// TwinCAT 3 PLC project PShEll_UniversalBlocks
// Title: PShEll Universal Blocks
// Company: Precision Systems Engineering
// Author: Control Systems Design Department
// ProjectVersion: 1.0.1.1
// Description: PSE Shell - Automation Software Development Kit
// ProgramVersion: 3.1.4023.0
// libraries:
//   CmpBitmapPool, * (System)
//   JS_MC_REF, * (Jenny Science AG)
//   Recipe Management, * (System)
//   Tc2_EtherCAT, * (Beckhoff Automation GmbH)
//   Tc2_IoFunctions, * (Beckhoff Automation GmbH)
//   Tc2_MC2, * (Beckhoff Automation GmbH)
//   Tc2_Standard, * (Beckhoff Automation GmbH)
//   Tc2_SUPS, * (Beckhoff Automation GmbH)
//   Tc2_System, * (Beckhoff Automation GmbH)
//   Tc2_SystemCX, * (Beckhoff Automation GmbH)
//   Tc2_TcpIp, * (Beckhoff Automation GmbH)
//   Tc2_Utilities, * (Beckhoff Automation GmbH)
//   Tc3_EventLogger, * (Beckhoff Automation GmbH)
//   Tc3_McCollisionAvoidance, * (Beckhoff Automation GmbH)
//   Tc3_McCompensations, * (Beckhoff Automation GmbH)
//   Tc3_McCoordinatedMotion, * (Beckhoff Automation GmbH)
//   Tc3_Module, * (Beckhoff Automation GmbH)
//   Tc3_XTS_Utility, * (Beckhoff Automation GmbH)
//   VisuDialogs, * (System)
//   VisuUserMgmt, * (System)
//   Tc2_Math,3.3.1.0,Beckhoff Automation GmbH
//   VisuSymbols,3.5.10.0,System
// project tree:
//   DUTs/Libs/Alarms/AlarmControler/ E_AlarmControlerState.TcDUT (not stored)
//   DUTs/Libs/Alarms/VisuEvents/ E_EventType.TcDUT (not stored), ST_BaseEvent.TcDUT (not stored), ST_Event.TcDUT (not stored)
//   DUTs/Libs/Axis/Universal Axis/ E_AxisJogDirection.TcDUT (not stored), E_AxisState.TcDUT (not stored), E_AxisStateInit.TcDUT (not stored), E_AxisStatePlcOpen.TcDUT (not stored)
//   DUTs/Libs/BowlFeeder/ E_BowlFeederUnitState.TcDUT, E_BowlFeederUnitStateInit.TcDUT
//   DUTs/Libs/Communication/TcpIp/ E_TcpIpDeviceState.TcDUT (not stored), E_TcpIpDeviceStateRecive.TcDUT (not stored), E_TcpIpDeviceStateSend.TcDUT (not stored), E_TcpIpServerStateRunning.TcDUT (not stored), ST_TcpBufferData.TcDUT (not stored)
//   DUTs/Libs/Cylinder/Universal Cylinder/ E_CylinderError.TcDUT (not stored), E_CylinderState.TcDUT (not stored), E_CylinderStateGo.TcDUT (not stored)
//   DUTs/Libs/Digital Devices/Digital Input/ E_DigitalInputExState.TcDUT (not stored)
//   DUTs/Libs/Digital Devices/Lamp Indicator/ E_LampState.TcDUT (not stored)
//   DUTs/Libs/Fixtures/UniversalFixture/ E_UniversalFixtureConnectionType.TcDUT (not stored), E_UniversalFixtureSampleResult.TcDUT (not stored), E_UniversalFixtureState.TcDUT (not stored), E_UniversalFixtureStateAbort.TcDUT (not stored), E_UniversalFixtureStateInit.TcDUT (not stored), E_UniversalFixtureStateMeasure.TcDUT (not stored), E_UniversalFixtureStateReset.TcDUT (not stored)
//   DUTs/Libs/Platform/Common/ ST_UniversalPlatform.TcDUT (not stored)
//   DUTs/Libs/Platform/Universal Machine/ E_MachineCtrlState.TcDUT (not stored)
//   DUTs/Libs/Platform/Universal Safety/ E_SafetyCtrlState.TcDUT (not stored)
//   DUTs/Libs/Platform/Universal Visu/ E_VisuCtrlAlarmControlState.TcDUT (not stored), E_VisuCtrlAxisImgType.TcDUT (not stored), E_VisuCtrlAxisJogMode.TcDUT (not stored), E_VisuCtrlCylinderImgType.TcDUT (not stored), E_VisuCtrlNavBarState.TcDUT (not stored), E_VisuCtrlPageState.TcDUT, E_VisuCtrlRecipeParameterType.TcDUT (not stored), E_VisuCtrlRecipesManagerState.TcDUT (not stored), E_VisuCtrlRobotImgType.TcDUT (not stored), E_VisuCtrlSingleAxisState.TcDUT (not stored), E_VisuCtrlSingleCylinderState.TcDUT (not stored), E_VisuCtrlSingleRobotState.TcDUT (not stored), E_VisuCtrUniversalMachineState.TcDUT (not stored), ST_VisuCtrlAxisFrame.TcDUT (not stored), ST_VisuCtrlCylinderFrame.TcDUT, ST_VisuCtrlFixtureFrame.TcDUT (not stored), ST_VisuCtrlInputFrame.TcDUT (not stored), ST_VisuCtrlOutputFrame.TcDUT (not stored), ST_VisuCtrlRecipeParameter.TcDUT (not stored), ST_VisuCtrlRecipesManager.TcDUT (not stored), ST_VisuCtrlRobotFrame.TcDUT (not stored), ST_VisuCtrlUnitFrame.TcDUT (not stored)
//   DUTs/Libs/Robots/Mitsubishi/CR800/EtherCAT Registers/ ST_CR800EthercatData.TcDUT (not stored)
//   DUTs/Libs/Robots/Mitsubishi/CR800/ E_CR800Error.TcDUT (not stored), ST_CR800UserDefinedArea.TcDUT (not stored)
//   DUTs/Libs/Robots/Mitsubishi/CR800/StateMachine/ E_CR800State.TcDUT (not stored), E_CR800StateAborting.TcDUT (not stored), E_CR800StateCommandExchange.TcDUT (not stored), E_CR800StateCyclePausing.TcDUT (not stored), E_CR800StateCycleStopping.TcDUT (not stored), E_CR800StateDoingRequest.TcDUT (not stored), E_CR800StateHoming.TcDUT (not stored), E_CR800StateInitializing.TcDUT (not stored), E_CR800StateSendPosition.TcDUT (not stored)
//   DUTs/Libs/Robots/Mitsubishi/ E_RobotActions.TcDUT (not stored), E_RobotSystemActions.TcDUT (not stored)
//   DUTs/Libs/SMC SI Unit/ ST_EX260_SEC1.TcDUT
//   DUTs/Libs/Utilities/CSV Data Exchanger/ E_CSVDataExchangerCountColumnsState.TcDUT (not stored), E_CSVDataExchangerInitState.TcDUT (not stored), E_CSVDataExchangerInsertIntoTableState.TcDUT (not stored), E_CSVDataExchangerSelectAllState.TcDUT (not stored), E_CSVDataExchangerSelectRowState.TcDUT (not stored), E_CSVDataExchangerSetNewPathState.TcDUT (not stored), E_CSVDataExchangerState.TcDUT (not stored), ST_CSV_Record.TcDUT (not stored)
//   DUTs/Libs/Utilities/File Logger/ E_FileLoggerAddLogsState.TcDUT (not stored), E_FileLoggerInitState.TcDUT (not stored), E_FileLoggerSetNewPathState.TcDUT (not stored), E_FileLoggerState.TcDUT (not stored)
//   DUTs/Libs/Utilities/Recipe Manager/ E_RecipesManagerReturns.TcDUT (not stored), E_RecipesManagerState.TcDUT (not stored), E_RecipesManagerStateBackup.TcDUT (not stored), E_RecipesManagerStateCreateRemove.TcDUT (not stored), E_RecipesManagerStateInit.TcDUT (not stored), E_RecipesManagerStateReload.TcDUT (not stored)
//   DUTs/Libs/Utilities/TXT Data Exchanger/ E_TXTDataExchangerAddLogsState.TcDUT (not stored), E_TXTDataExchangerInitState.TcDUT (not stored), E_TXTDataExchangerSearchForFileState.TcDUT (not stored), E_TXTDataExchangerSetNewPathState.TcDUT (not stored), E_TXTDataExchangerState.TcDUT (not stored)
//   DUTs/Libs/Vision/Cognex/ E_CognexCameraGetConnectionStatus.TcDUT (not stored), E_CognexCameraGetExprStatus.TcDUT (not stored), E_CognexCameraGetFileListStatus.TcDUT (not stored), E_CognexCameraGetFileStatus.TcDUT (not stored), E_CognexCameraGetJobStatus.TcDUT (not stored), E_CognexCameraGetOnlineStatus.TcDUT (not stored), E_CognexCameraGetPositionState.TcDUT (not stored), E_CognexCameraGetPositionStatus.TcDUT (not stored), E_CognexCameraGetValueEasyBuilderStatus.TcDUT (not stored), E_CognexCameraGetValueSpreadsheetStatus.TcDUT (not stored), E_CognexCameraGetValuesState.TcDUT (not stored), E_CognexCameraGetValuesStatus.TcDUT (not stored), E_CognexCameraGetValueStatus.TcDUT (not stored), E_CognexCameraImageTriggerStatus.TcDUT (not stored), E_CognexCameraInitState.TcDUT (not stored), E_CognexCameraLoadFileStatus.TcDUT (not stored), E_CognexCameraMethodState.TcDUT (not stored), E_CognexCameraPutLiveStatus.TcDUT (not stored), E_CognexCameraPutPortnumStatus.TcDUT (not stored), E_CognexCameraPutTimeoutStatus.TcDUT (not stored), E_CognexCameraPutUpdateStatus.TcDUT (not stored), E_CognexCameraPutWatchStatus.TcDUT (not stored), E_CognexCameraResetSystemStatus.TcDUT (not stored), E_CognexCameraSetJobStatus.TcDUT (not stored), E_CognexCameraSetOnlineStatus.TcDUT (not stored), E_CognexCameraState.TcDUT (not stored), E_CognexCameraStoreFileStatus.TcDUT (not stored)
//   DUTs/Machine/Machine Control/Batch/ ST_BatchData.TcDUT, ST_BatchPerformacne.TcDUT
//   DUTs/Machine/Machine Control/ E_MachineCtrlStateAbort.TcDUT, E_MachineCtrlStateAuto.TcDUT, E_MachineCtrlStateAutoAOI.TcDUT, E_MachineCtrlStateInit.TcDUT, E_MachineCtrlStateManualToAuto.TcDUT, E_MachineCtrlStateUninitialized.TcDUT
//   DUTs/Machine/Machine Control/Internal/ E_GoldenSampleMeasurementState.TcDUT, E_RotaryTableState.TcDUT
//   DUTs/Machine/Shell API/ ST_Shell.TcDUT (not stored), ST_ShellFlags.TcDUT (not stored), ST_ShellPlatform.TcDUT, ST_ShellRecipeData.TcDUT (not stored)
//   DUTs/Machine/Visu Control/ E_VisuCtrlInitializingPopUpFrameSelector.TcDUT, E_VisuCtrlUninitializedFrameSelector.TcDUT, ST_InitializationFrame.TcDUT, ST_UninitializedSetupFrame.TcDUT, ST_UninitializedStartUpFrame.TcDUT
//   / GlobalTextList.TcGTLO, PlcTask.TcTTO, Visualization Manager.TcVMO (not stored), VISU_TASK.TcTTO
//   GVLs/ GVL.TcGVL
//   POUs/Libs/0_Checks/Checks/ CheckBounds.TcPOU (not stored), CheckDivDInt.TcPOU (not stored), CheckDivLInt.TcPOU (not stored), CheckDivLReal.TcPOU (not stored), CheckDivReal.TcPOU (not stored), CheckPointer.TcPOU (not stored), CheckRangeSigned.TcPOU (not stored), CheckRangeUnsigned.TcPOU (not stored), P_Checks.TcPOU (not stored)
//   POUs/Libs/0_Checks/ GVL_Checks.TcGVL (not stored)
//   POUs/Libs/Alarms/AlarmControler/ FB_AlarmControler.TcPOU (not stored), I_AlarmControler.TcIO (not stored)
//   POUs/Libs/Alarms/VisuEvents/ FB_VisuEventsHandling.TcPOU, LDT_TO_STRING.TcPOU (not stored)
//   POUs/Libs/Analog Devices/Analog Device/ FB_AnalogDevice.TcPOU, I_AnalogDevice.TcIO
//   POUs/Libs/Analog Devices/Analog Output/ FB_AnalogOutput.TcPOU, I_AnalogOutput.TcIO
//   POUs/Libs/Axis/ FB_AxisServo.TcPOU (not stored), FB_UniversalAxis.TcPOU (not stored), I_UniversalAxis.TcIO (not stored)
//   POUs/Libs/Bowl Feeder/ FB_BowlFeeder.TcPOU, I_BowlFeeder.TcIO
//   POUs/Libs/Communication/TcpIp/ FUN_StringToTcpBufferData.TcPOU (not stored), FUN_TcpBufferDataToString.TcPOU (not stored)
//   POUs/Libs/Communication/TcpIp/Tcp Buffer/ FB_TcpBuffer.TcPOU (not stored)
//   POUs/Libs/Communication/TcpIp/Tcp Client/ FB_TcpClient.TcPOU (not stored)
//   POUs/Libs/Communication/TcpIp/Tcp Device/ FB_TcpDevice.TcPOU (not stored), I_TcpDevice.TcIO (not stored)
//   POUs/Libs/Communication/TcpIp/Tcp Server/ FB_TcpServer.TcPOU (not stored)
//   POUs/Libs/Cylinder/Double Coil Cylinder/ FB_DoubleCoilCylinder.TcPOU (not stored), FB_DoubleCoilCylinder2.TcPOU (not stored)
//   POUs/Libs/Cylinder/Single Coil Cylinder/ FB_SingleCoilCylinder.TcPOU (not stored), FB_SingleCoilCylinder2.TcPOU (not stored)
//   POUs/Libs/Cylinder/Universal Cylinder/ FB_UniversalCylinder.TcPOU (not stored), I_UniversalCylinder.TcIO (not stored)
//   POUs/Libs/Digital Devices/Digital Device/ FB_DigitalDevice.TcPOU (not stored), I_DigitalDevice.TcIO (not stored)
//   POUs/Libs/Digital Devices/Digital Input/ FB_DigitalInput.TcPOU (not stored), FB_DigitalInputExt.TcPOU (not stored), I_DigitalInput.TcIO (not stored)
//   POUs/Libs/Digital Devices/Digital Output/ FB_DigitalOutput.TcPOU (not stored), I_DigitalOutput.TcIO (not stored)
//   POUs/Libs/Digital Devices/Lamp Indicator/ FB_Lamp.TcPOU (not stored), I_Lamp.TcIO (not stored)
//   POUs/Libs/Fixtures/ FB_UniversalFixture.TcPOU (not stored), I_UniversalFixture.TcIO (not stored)
//   POUs/Libs/Platform/Universal Machine/ FB_UniversalMachine.TcPOU (not stored), I_UniversalMachine.TcIO (not stored)
//   POUs/Libs/Platform/Universal Safety/ FB_UniversalSafety.TcPOU (not stored), I_UniversalSafety.TcIO (not stored)
//   POUs/Libs/Platform/Universal Visu/ FB_UniversalVisu.TcPOU, F_CloseDialog.TcPOU (not stored), F_OpenDialog.TcPOU (not stored)
//   POUs/Libs/Robots/Mitsubishi/ FB_CR800EtherCAT.TcPOU, I_CR800EtherCAT.TcIO (not stored)
//   POUs/Libs/Utilities/Beckhoff UPS/CX2xxx/ FB_UpsCx2xxx.TcPOU (not stored)
//   POUs/Libs/Utilities/Beckhoff UPS/CX5xxx/ FB_UpsCx50xx.TcPOU (not stored), FB_UpsCx51xx.TcPOU (not stored), FB_UpsCx5xxx.TcPOU (not stored), I_BeckhoffUpsCX5xxx.TcIO (not stored)
//   POUs/Libs/Utilities/Beckhoff UPS/Universal CX/ FB_UniversalCxUps.TcPOU (not stored), I_UniversalCxUps.TcIO (not stored)
//   POUs/Libs/Utilities/CSV Data Exchanger/ FB_CSVDataExchanger.TcPOU (not stored), I_CSVDataExchanger.TcIO (not stored)
//   POUs/Libs/Utilities/ FB_DataSetFifo.TcPOU (excluded from build), FB_DataSetFifo_1.TcPOU
//   POUs/Libs/Utilities/File Logger/ FB_FileLogger.TcPOU (not stored), I_FileLogger.TcIO (not stored)
//   POUs/Libs/Utilities/Math/ FUN_Ceil.TcPOU (not stored)
//   POUs/Libs/Utilities/Recipes Manager/ FB_RecipeParameter.TcPOU (not stored), FB_RecipesControler.TcPOU (not stored), I_RecipeParameter.TcIO (not stored), I_RecipesManager.TcIO (not stored)
//   POUs/Libs/Utilities/StringMerge/ FUN_MergeLongStrings10.TcPOU (not stored), FUN_MergeStrings10.TcPOU (not stored), FUN_MergeStrings3.TcPOU (not stored), FUN_MergeStrings4.TcPOU (not stored), FUN_MergeStrings5.TcPOU (not stored), FUN_MergeStrings6.TcPOU (not stored)
//   POUs/Libs/Utilities/Systemtime to String/ FUN_TimestructToDate.TcPOU (not stored), FUN_TimestructToTime.TcPOU (not stored)
//   POUs/Libs/Utilities/TXT Data Exchanger/ FB_TXTDataExchanger.TcPOU (not stored), I_TXTDataExchanger.TcIO (not stored)
//   POUs/Libs/Vision/Cognex/ FB_CognexCamera.TcPOU (not stored), I_CognexCamera.TcIO (not stored)
//   POUs/Machine/ FB_MachineControl.TcPOU, FB_MachineSafety.TcPOU, FB_VisuControl.TcPOU, I_MachineControl.TcIO, ST_VisuCtrlBowlFeeder.TcDUT
//   POUs/Machine/Module/Robot/ E_AOIRobotActions.TcDUT, E_AOIRobotState.TcDUT, E_AOIRobotStateAbort.TcDUT, E_AOIRobotStateInit.TcDUT, E_EtherCATStatusCheck.TcDUT, FB_Robot.TcPOU, I_AOIRobot.TcIO
//   POUs/Machine/Module/RTCVision/ E_RTCCameraInitState.TcDUT, E_RTCCameraMethodState.TcDUT, E_RTCCameraState.TcDUT, E_VisionJob.TcDUT, E_VisionResult.TcDUT, FB_DoubleTrigger.TcPOU, FB_RTCVision.TcPOU, I_RTCVision.TcIO (excluded from build)
//   POUs/Machine/Visu Control/ F_CloseDialog_1.TcPOU (not stored), F_OpenDialog_1.TcPOU (not stored)
//   POUs/PRG/ PRG_AlarmControl.TcPOU, PRG_FB_BowlFeeder.TcPOU (excluded from build), PRG_MachineControl.TcPOU, PRG_MachineSafety.TcPOU, PRG_RecipesManager.TcPOU (not stored), PRG_VisuControl.TcPOU
//   VISUs/Alarms/ EventTable.TcVIS (not stored), EventTableNew.TcVIS (not stored), SingleEvent.TcVIS (not stored)
//   VISUs/Alarms/Image Pools/ IP_EventSeverity.TcIPO (not stored), IP_EventType.TcIPO (not stored)
//   VISUs/Alarms/Text Lists/ TL_EventServerity.TcTLO (not stored), TL_EventType.TcTLO (not stored)
//   VISUs/Headers/ Header.TcVIS, HeaderWinCE.TcVIS (not stored)
//   VISUs/Headers/Image Pools/ IPHeader.TcIPO (not stored)
//   VISUs/Headers/Text Lists/ TL_HeaderMachineState.TcTLO (not stored)
//   VISUs/ Main.TcVIS
//   VISUs/Manual/Image Pools/ IPAxis.TcIPO (not stored), IPCylinder.TcIPO (not stored), IPRobots.TcIPO (not stored)
//   VISUs/Manual/ SingleAxis.TcVIS, SingleFixture.TcVIS (not stored), SingleAxisJogInching.TcVIS (not stored), SingleAxisJogContinous.TcVIS (not stored), SingleAxisJogInchingModulo.TcVIS (not stored), SingleAxisJogStandardSlow.TcVIS (not stored), SingleAxisJogStandardFlast.TcVIS (not stored), SingleCylinder.TcVIS (not stored), SingleDigitalInput.TcVIS, SingleRobot.TcVIS (not stored), SingleSafeOutput.TcVIS (not stored) (excluded from build), SingleSafeInput.TcVIS (not stored) (excluded from build), SingleDigitalOutput.TcVIS (not stored)
//   VISUs/Manual/Text Lists/ TL_ModeSwitchState.TcTLO (not stored), TL_SingleAxisJogMode.TcTLO (not stored), TL_SingleCylinderState.TcTLO (not stored), TL_SingleAxisState.TcTLO (not stored), TL_SingleRobotState.TcTLO (not stored)
//   VISUs/Navigation/ NavBarAuto.TcVIS, NavBarAuxilary.TcVIS, NavBarEmpty.TcVIS (not stored), NavBarInitializing.TcVIS (not stored), NavBarManual.TcVIS, NavBarUninitialized.TcVIS, NavBarUtilities.TcVIS (not stored)
//   VISUs/Pages/Auto/ AOIBowlFeederFrame.TcVIS, AOIBatchPerformanceFrame.TcVIS, AOIHeaderFrame.TcVIS (excluded from build), AOIHeaderKeySwitchFrame.TcVIS (excluded from build), AOIBatchDataFrame.TcVIS (excluded from build), AOISortStationFrame.TcVIS, PageAuto.TcVIS, ST_SortStationParam.TcDUT
//   VISUs/Pages/Initializing/ InitializingDoorLockOpen.TcVIS, InitializingEStopActive.TcVIS, InitializingFixtureConnectionFailed.TcVIS (excluded from build), InitializingNoFixturesAvailable.TcVIS (excluded from build), InitializingRotaryTablePlaceTrayDialog.TcVIS (excluded from build), InitializingStartSafetySystem.TcVIS, InitializingTrayfeederCourtainBroken.TcVIS (excluded from build), InitializingTrayfeederInterupted.TcVIS (excluded from build), PageInitializing.TcVIS
//   VISUs/Pages/ PageAborting.TcVIS (not stored), PageAlarms.TcVIS, PageManualCylinders.TcVIS (not stored), PageManualRobots.TcVIS (not stored), PageManualInputs.TcVIS (not stored), PageManualAxis.TcVIS (not stored), PageManualOutputs.TcVIS (not stored), PageManualSafety.TcVIS (not stored) (excluded from build), PageReadyInitialized.TcVIS (not stored), PageRecipesManager.TcVIS (not stored), PageReset.TcVIS (not stored), PageSwitchMode.TcVIS (not stored)
//   VISUs/Pages/Uninitialized/ PageUninitialized.TcVIS, UninitializedSetupFrame.TcVIS, UninitializedStartUpFrame.TcVIS
//   VISUs/Recipes/ SingleRecipesParameterTypeBool.TcVIS (not stored), SingleRecipesParameterTypeInteger.TcVIS (not stored), SingleRecipesParameterTypeReal.TcVIS (not stored), SingleRecipesParameterTypeString.TcVIS (not stored)
//   VISUs/Recipes/Text Lists/ TL_RecipesManagerReturns.TcTLO (not stored), TL_RecipesManagerStatus.TcTLO (not stored)
// real-time tasks:
//   TASK PlcTask: cycle T#10ms, priority 20, ADS port 350
//   TASK VISU_TASK: cycle T#100000us, priority 30, ADS port 351
// motion (NC):
//   TASK NC-Task 1 SAF: cycle T#2ms, priority 4, ADS port 501
//   TASK NC-Task 1 SVB: cycle T#10ms, priority 8, ADS port 511
//   AXIS Rotary Table (id 2)
//     General: UnitName=°
//     OtherSettings: AllowMotionCmdToSlave=true
//     encoder EncType=19
//       EncPara: ScaleFactorNumerator=72, ScaleFactorDenominator=10000, MaxCount=#xffffffff
//         Inc: RefSearchInverse=true, RefSyncInverse=false
//     drive DrvType=16
//       DrvPara: MaxCount=#xffffffff, DriveControlDWord=#x00020000
//         Analog: TorqueSetpointScale=10, ScaleFactorActTorque=0.1
//         TimeComp: TaskDelayCycles=1
//     controller CtrType=1
//       CtrPara: PriorControlFactor=1
//         Observer: BandWidth=20
// I/O:
//   DEVICE Device 1 (EtherCAT), AmsNetId 5.127.48.56.2.1
//     Term 1 (EK1200) [EK1200-5000 EtherCAT Power supply (2A E-Bus)]
//       Term 2 (EL6900) [EL6900, TwinSAFE PLC]
//       Term 3 (EL6070-0033) [EL6070-0033 1Ch. Licence key terminal, individual licences]
//       Term 4 (EL1904) [EL1904, 4 Ch. Safety Input 24V, TwinSAFE]
//         modules: Module 1 (FSOES)
//       Term 5 (EL1114) [EL1114 4Ch. Dig. Input 24V, 10µs, Sensor Power]
//       Term 6 (EL1904) [EL1904, 4 Ch. Safety Input 24V, TwinSAFE]
//         modules: Module 1 (FSOES)
//       Term 7 (EL2004) [EL2004 4Ch. Dig. Output 24V, 0.5A]
//       Term 8 (EL2904) [EL2904, 4 Ch. Safety Output 24V, 0.5A, TwinSAFE]
//         modules: Module 1 (FSOES), Module 2 (DO)
//       Term 9 (EL1114) [EL1114 4Ch. Dig. Input 24V, 10µs, Sensor Power]
//       Term 10 (EL4004) [EL4004 4Ch. Ana. Output 0-10V, 12bit]
//       Term 11 (EL1904) [EL1904, 4 Ch. Safety Input 24V, TwinSAFE]
//         modules: Module 1 (FSOES)
//       Term 12 (EL2004) [EL2004 4Ch. Dig. Output 24V, 0.5A]
//       Term 13 (EL2004) [EL2004 4Ch. Dig. Output 24V, 0.5A]
//       Term 14 (EL9410) [EL9410 E-Bus Power Supplier  (Diagnostics)]
//       Term 15 (EL1904) [EL1904, 4 Ch. Safety Input 24V, TwinSAFE]
//         modules: Module 1 (FSOES)
//       Term 16 (EL2004) [EL2004 4Ch. Dig. Output 24V, 0.5A]
//       Term 17 (EL2004) [EL2004 4Ch. Dig. Output 24V, 0.5A]
//       Term 18 (EL2904) [EL2904, 4 Ch. Safety Output 24V, 0.5A, TwinSAFE]
//         modules: Module 1 (FSOES), Module 2 (DO)
//       Term 19 (EL1114) [EL1114 4Ch. Dig. Input 24V, 10µs, Sensor Power]
//       Term 20 (EK1122) [EK1122 2 port EtherCAT junction]
//         Box 21 (CompactCom 40 EtherCAT) [CompactCom 40 EtherCAT]
//           modules: Module 1 (4 Stations:CR800 GPIO_REG_IF)
//         Drive 22 (Ezi-SERVO2 EtherCAT) [Ezi-SERVO2 EtherCAT]
//         Box 23 (EX260-SEC1) [EX260-SEC1 EtherCAT SI Unit (32DO_PNP) Rev1.2]
// variable links:
//   NC-Task 1 SAF/Axes/Rotary Table <-> Device 1 (EtherCAT)/Term 1 (EK1200)/Term 20 (EK1122)/Drive 22 (Ezi-SERVO2 EtherCAT)
//     Drive/Inputs/In/nDcOutputTime <-> InfoData/DcOutputShift
//     Drive/Inputs/In/nState1 <-> CSP Inputs/Status Word
//     Drive/Inputs/In/nState2 <-> CSP Inputs/Status Word @bit 8
//     Drive/Inputs/In/nState4 @bit 1 <-> WcState/InputToggle
//     Drive/Inputs/In/nState4 <-> WcState/WcState
//     Drive/Outputs/Out/nCtrl1 <-> CSP Outputs/Control Word
//     Drive/Outputs/Out/nCtrl2 <-> CSP Outputs/Control Word @bit 8
//     Drive/Outputs/Out/nDataOut1 <-> CSP Outputs/Target Position
//     Enc/Inputs/In/nDataIn1 <-> CSP Inputs/Position Actual Value
//     Enc/Inputs/In/nDataIn3 <-> CSP Inputs/Touch probe 1 positive value
//     Enc/Inputs/In/nDataIn5 <-> CSP Inputs/Touch probe 2 positive value
//     Enc/Inputs/In/nDcInputTime <-> InfoData/DcInputShift
//     Enc/Inputs/In/nState4 @bit 1 <-> WcState/InputToggle
//     Enc/Inputs/In/nState4 <-> WcState/WcState
//     Enc/Inputs/In/nState5 <-> CSP Inputs/Touch probe status
//     Enc/Inputs/In/nState6 <-> CSP Inputs/Touch probe status @bit 8
//     Enc/Outputs/Out/nCtrl5 <-> CSP Outputs/Touch probe function
//     Enc/Outputs/Out/nCtrl6 <-> CSP Outputs/Touch probe function @bit 8
//   PShEll_UniversalBlocks/PShEll_UniversalBlocks Instance <-> Device 1 (EtherCAT)/Term 1 (EK1200)/Term 10 (EL4004)
//     PlcTask Outputs/PRG_MachineControl.fbMachineControler.fbBowlFeeder._aoSetpoint.intAnalogOut <-> AO Outputs Channel 1/Analog output
//   PShEll_UniversalBlocks/PShEll_UniversalBlocks Instance <-> Device 1 (EtherCAT)/Term 1 (EK1200)/Term 13 (EL2004)
//     PlcTask Outputs/PRG_MachineControl.fbMachineControler.fbBowlFeeder.doEnable.bOut <-> Channel 1/Output
//     PlcTask Outputs/PRG_MachineControl.fbMachineControler.fbRobot.doRobotModeSwitch.bOut <-> Channel 3/Output
//   PShEll_UniversalBlocks/PShEll_UniversalBlocks Instance <-> Device 1 (EtherCAT)/Term 1 (EK1200)/Term 16 (EL2004)
//     PlcTask Outputs/PRG_MachineControl.fbMachineControler.doTriggerCam{1..4}.doCam.bOut <-> Channel {1..4}/Output  (4 links)
//   PShEll_UniversalBlocks/PShEll_UniversalBlocks Instance <-> Device 1 (EtherCAT)/Term 1 (EK1200)/Term 17 (EL2004)
//     PlcTask Outputs/PRG_MachineControl.fbMachineControler.doTriggerCam5.doCam.bOut <-> Channel 1/Output
//     PlcTask Outputs/PRG_MachineControl.fbMachineControler.doTriggerCam6.doCam.bOut <-> Channel 2/Output
//     PlcTask Outputs/PRG_MachineControl.fbMachineControler.doTriggerCam7.doCam.bOut <-> Channel 3/Output
//   PShEll_UniversalBlocks/PShEll_UniversalBlocks Instance <-> Device 1 (EtherCAT)/Term 1 (EK1200)/Term 19 (EL1114)
//     PlcTask Inputs/PRG_MachineControl.fbMachineControler.diProductPresenceRobot.bIn <-> Channel 4/Input
//     PlcTask Inputs/PRG_MachineControl.fbMachineControler.fbBowlFeeder.diStatusRelay.bIn <-> Channel 3/Input
//   PShEll_UniversalBlocks/PShEll_UniversalBlocks Instance <-> Device 1 (EtherCAT)/Term 1 (EK1200)/Term 20 (EK1122)/Box 21 (CompactCom 40 EtherCAT)
//     PlcTask Inputs/PRG_MachineControl.fbMachineControler.fbRobot.fbCR800.stCR800EthercatData.arrRegistersInput[6000] <-> Module 1 (4 Stations:CR800 GPIO_REG_IF)/Tx PDO (4 Sta.)/RWr(6000)
//     PlcTask Inputs/PRG_MachineControl.fbMachineControler.fbRobot.fbCR800.stCR800EthercatData.arrRegistersInput[6001] <-> Module 1 (4 Stations:CR800 GPIO_REG_IF)/Tx PDO (4 Sta.)/RWr(6001)
//     PlcTask Inputs/PRG_MachineControl.fbMachineControler.fbRobot.fbCR800.stCR800EthercatData.arrRegistersInput[6002] <-> Module 1 (4 Stations:CR800 GPIO_REG_IF)/Tx PDO (4 Sta.)/RWr(6002)
//     PlcTask Inputs/PRG_MachineControl.fbMachineControler.fbRobot.fbCR800.stCR800EthercatData.arrRegistersInput[6003] <-> Module 1 (4 Stations:CR800 GPIO_REG_IF)/Tx PDO (4 Sta.)/RWr(6003)
//     PlcTask Inputs/PRG_MachineControl.fbMachineControler.fbRobot.fbCR800.stCR800EthercatData.arrRegistersInput[6004] <-> Module 1 (4 Stations:CR800 GPIO_REG_IF)/Tx PDO (4 Sta.)/RWr(6004)
//     PlcTask Inputs/PRG_MachineControl.fbMachineControler.fbRobot.fbCR800.stCR800EthercatData.arrRegistersInput[6005] <-> Module 1 (4 Stations:CR800 GPIO_REG_IF)/Tx PDO (4 Sta.)/RWr(6005)
//     PlcTask Inputs/PRG_MachineControl.fbMachineControler.fbRobot.fbCR800.stCR800EthercatData.arrRegistersInput[6006] <-> Module 1 (4 Stations:CR800 GPIO_REG_IF)/Tx PDO (4 Sta.)/RWr(6006)
//     PlcTask Inputs/PRG_MachineControl.fbMachineControler.fbRobot.fbCR800.stCR800EthercatData.arrRegistersInput[6007] <-> Module 1 (4 Stations:CR800 GPIO_REG_IF)/Tx PDO (4 Sta.)/RWr(6007)
//     PlcTask Inputs/PRG_MachineControl.fbMachineControler.fbRobot.fbCR800.stCR800EthercatData.arrRegistersInput[6008] <-> Module 1 (4 Stations:CR800 GPIO_REG_IF)/Tx PDO (4 Sta.)/RWr(6008)
//     PlcTask Inputs/PRG_MachineControl.fbMachineControler.fbRobot.fbCR800.stCR800EthercatData.arrRegistersInput[6009] <-> Module 1 (4 Stations:CR800 GPIO_REG_IF)/Tx PDO (4 Sta.)/RWr(6009)
//     PlcTask Inputs/PRG_MachineControl.fbMachineControler.fbRobot.fbCR800.stCR800EthercatData.arrRegistersInput[6010] <-> Module 1 (4 Stations:CR800 GPIO_REG_IF)/Tx PDO (4 Sta.)/RWr(6010)
//     PlcTask Inputs/PRG_MachineControl.fbMachineControler.fbRobot.fbCR800.stCR800EthercatData.arrRegistersInput[6011] <-> Module 1 (4 Stations:CR800 GPIO_REG_IF)/Tx PDO (4 Sta.)/RWr(6011)
//     PlcTask Inputs/PRG_MachineControl.fbMachineControler.fbRobot.fbCR800.stCR800EthercatData.arrRegistersInput[6012] <-> Module 1 (4 Stations:CR800 GPIO_REG_IF)/Tx PDO (4 Sta.)/RWr(6012)
//     PlcTask Inputs/PRG_MachineControl.fbMachineControler.fbRobot.fbCR800.stCR800EthercatData.arrRegistersInput[6013] <-> Module 1 (4 Stations:CR800 GPIO_REG_IF)/Tx PDO (4 Sta.)/RWr(6013)
//     PlcTask Inputs/PRG_MachineControl.fbMachineControler.fbRobot.fbCR800.stCR800EthercatData.arrRegistersInput[6014] <-> Module 1 (4 Stations:CR800 GPIO_REG_IF)/Tx PDO (4 Sta.)/RWr(6014)
//     PlcTask Inputs/PRG_MachineControl.fbMachineControler.fbRobot.fbCR800.stCR800EthercatData.arrRegistersInput[6015] <-> Module 1 (4 Stations:CR800 GPIO_REG_IF)/Tx PDO (4 Sta.)/RWr(6015)
//     PlcTask Inputs/PRG_MachineControl.fbMachineControler.fbRobot.fbCR800.stCR800EthercatData.arrRegistersInput[6016] <-> Module 1 (4 Stations:CR800 GPIO_REG_IF)/Tx PDO (4 Sta.)/RWr(6016)
//     PlcTask Inputs/PRG_MachineControl.fbMachineControler.fbRobot.fbCR800.stCR800EthercatData.arrRegistersInput[6017] <-> Module 1 (4 Stations:CR800 GPIO_REG_IF)/Tx PDO (4 Sta.)/RWr(6017)
//     PlcTask Inputs/PRG_MachineControl.fbMachineControler.fbRobot.fbCR800.stCR800EthercatData.arrRegistersInput[6018] <-> Module 1 (4 Stations:CR800 GPIO_REG_IF)/Tx PDO (4 Sta.)/RWr(6018)
//     PlcTask Inputs/PRG_MachineControl.fbMachineControler.fbRobot.fbCR800.stCR800EthercatData.arrRegistersInput[6019] <-> Module 1 (4 Stations:CR800 GPIO_REG_IF)/Tx PDO (4 Sta.)/RWr(6019)
//     PlcTask Inputs/PRG_MachineControl.fbMachineControler.fbRobot.fbCR800.stCR800EthercatData.arrRegistersInput[6020] <-> Module 1 (4 Stations:CR800 GPIO_REG_IF)/Tx PDO (4 Sta.)/RWr(6020)
//     PlcTask Inputs/PRG_MachineControl.fbMachineControler.fbRobot.fbCR800.stCR800EthercatData.arrRegistersInput[6021] <-> Module 1 (4 Stations:CR800 GPIO_REG_IF)/Tx PDO (4 Sta.)/RWr(6021)
//     PlcTask Inputs/PRG_MachineControl.fbMachineControler.fbRobot.fbCR800.stCR800EthercatData.arrRegistersInput[6022] <-> Module 1 (4 Stations:CR800 GPIO_REG_IF)/Tx PDO (4 Sta.)/RWr(6022)
//     PlcTask Inputs/PRG_MachineControl.fbMachineControler.fbRobot.fbCR800.stCR800EthercatData.arrRegistersInput[6023] <-> Module 1 (4 Stations:CR800 GPIO_REG_IF)/Tx PDO (4 Sta.)/RWr(6023)
//     PlcTask Inputs/PRG_MachineControl.fbMachineControler.fbRobot.fbCR800.stCR800EthercatData.arrRegistersInput[6024] <-> Module 1 (4 Stations:CR800 GPIO_REG_IF)/Tx PDO (4 Sta.)/RWr(6024)
//     PlcTask Inputs/PRG_MachineControl.fbMachineControler.fbRobot.fbCR800.stCR800EthercatData.arrRegistersInput[6025] <-> Module 1 (4 Stations:CR800 GPIO_REG_IF)/Tx PDO (4 Sta.)/RWr(6025)
//     PlcTask Inputs/PRG_MachineControl.fbMachineControler.fbRobot.fbCR800.stCR800EthercatData.arrRegistersInput[6026] <-> Module 1 (4 Stations:CR800 GPIO_REG_IF)/Tx PDO (4 Sta.)/RWr(6026)
//     PlcTask Inputs/PRG_MachineControl.fbMachineControler.fbRobot.fbCR800.stCR800EthercatData.arrRegistersInput[6027] <-> Module 1 (4 Stations:CR800 GPIO_REG_IF)/Tx PDO (4 Sta.)/RWr(6027)
//     PlcTask Inputs/PRG_MachineControl.fbMachineControler.fbRobot.fbCR800.stCR800EthercatData.arrRegistersInput[6028] <-> Module 1 (4 Stations:CR800 GPIO_REG_IF)/Tx PDO (4 Sta.)/RWr(6028)
//     PlcTask Inputs/PRG_MachineControl.fbMachineControler.fbRobot.fbCR800.stCR800EthercatData.arrRegistersInput[6029] <-> Module 1 (4 Stations:CR800 GPIO_REG_IF)/Tx PDO (4 Sta.)/RWr(6029)
//     PlcTask Inputs/PRG_MachineControl.fbMachineControler.fbRobot.fbCR800.stCR800EthercatData.arrRegistersInput[6030] <-> Module 1 (4 Stations:CR800 GPIO_REG_IF)/Tx PDO (4 Sta.)/RWr(6030)
//     PlcTask Inputs/PRG_MachineControl.fbMachineControler.fbRobot.fbCR800.stCR800EthercatData.arrRegistersInput[6031] <-> Module 1 (4 Stations:CR800 GPIO_REG_IF)/Tx PDO (4 Sta.)/RWr(6031)
//     PlcTask Inputs/PRG_MachineControl.fbMachineControler.fbRobot.fbCR800.stCR800EthercatData.arrRegistersInput[6032] <-> Module 1 (4 Stations:CR800 GPIO_REG_IF)/Tx PDO (4 Sta.)/RWr(6032)
//     PlcTask Inputs/PRG_MachineControl.fbMachineControler.fbRobot.fbCR800.stCR800EthercatData.arrRegistersInput[6033] <-> Module 1 (4 Stations:CR800 GPIO_REG_IF)/Tx PDO (4 Sta.)/RWr(6033)
//     PlcTask Inputs/PRG_MachineControl.fbMachineControler.fbRobot.fbCR800.stCR800EthercatData.arrRegistersInput[6034] <-> Module 1 (4 Stations:CR800 GPIO_REG_IF)/Tx PDO (4 Sta.)/RWr(6034)
//     PlcTask Inputs/PRG_MachineControl.fbMachineControler.fbRobot.fbCR800.stCR800EthercatData.arrRegistersInput[6035] <-> Module 1 (4 Stations:CR800 GPIO_REG_IF)/Tx PDO (4 Sta.)/RWr(6035)
//     PlcTask Inputs/PRG_MachineControl.fbMachineControler.fbRobot.fbCR800.stCR800EthercatData.arrRegistersInput[6036] <-> Module 1 (4 Stations:CR800 GPIO_REG_IF)/Tx PDO (4 Sta.)/RWr(6036)
//     PlcTask Inputs/PRG_MachineControl.fbMachineControler.fbRobot.fbCR800.stCR800EthercatData.arrRegistersInput[6037] <-> Module 1 (4 Stations:CR800 GPIO_REG_IF)/Tx PDO (4 Sta.)/RWr(6037)
//     PlcTask Inputs/PRG_MachineControl.fbMachineControler.fbRobot.fbCR800.stCR800EthercatData.arrRegistersInput[6038] <-> Module 1 (4 Stations:CR800 GPIO_REG_IF)/Tx PDO (4 Sta.)/RWr(6038)
//     PlcTask Inputs/PRG_MachineControl.fbMachineControler.fbRobot.fbCR800.stCR800EthercatData.arrRegistersInput[6039] <-> Module 1 (4 Stations:CR800 GPIO_REG_IF)/Tx PDO (4 Sta.)/RWr(6039)
//     PlcTask Inputs/PRG_MachineControl.fbMachineControler.fbRobot.fbCR800.stCR800EthercatData.arrRegistersInput[6040] <-> Module 1 (4 Stations:CR800 GPIO_REG_IF)/Tx PDO (4 Sta.)/RWr(6040)
//     PlcTask Inputs/PRG_MachineControl.fbMachineControler.fbRobot.fbCR800.stCR800EthercatData.arrRegistersInput[6041] <-> Module 1 (4 Stations:CR800 GPIO_REG_IF)/Tx PDO (4 Sta.)/RWr(6041)
//     PlcTask Inputs/PRG_MachineControl.fbMachineControler.fbRobot.fbCR800.stCR800EthercatData.arrRegistersInput[6042] <-> Module 1 (4 Stations:CR800 GPIO_REG_IF)/Tx PDO (4 Sta.)/RWr(6042)
//     PlcTask Inputs/PRG_MachineControl.fbMachineControler.fbRobot.fbCR800.stCR800EthercatData.arrRegistersInput[6043] <-> Module 1 (4 Stations:CR800 GPIO_REG_IF)/Tx PDO (4 Sta.)/RWr(6043)
//     PlcTask Inputs/PRG_MachineControl.fbMachineControler.fbRobot.fbCR800.stCR800EthercatData.arrRegistersInput[6044] <-> Module 1 (4 Stations:CR800 GPIO_REG_IF)/Tx PDO (4 Sta.)/RWr(6044)
//     PlcTask Inputs/PRG_MachineControl.fbMachineControler.fbRobot.fbCR800.stCR800EthercatData.arrRegistersInput[6045] <-> Module 1 (4 Stations:CR800 GPIO_REG_IF)/Tx PDO (4 Sta.)/RWr(6045)
//     PlcTask Inputs/PRG_MachineControl.fbMachineControler.fbRobot.fbCR800.stCR800EthercatData.arrRegistersInput[6046] <-> Module 1 (4 Stations:CR800 GPIO_REG_IF)/Tx PDO (4 Sta.)/RWr(6046)
//     PlcTask Inputs/PRG_MachineControl.fbMachineControler.fbRobot.fbCR800.stCR800EthercatData.arrRegistersInput[6047] <-> Module 1 (4 Stations:CR800 GPIO_REG_IF)/Tx PDO (4 Sta.)/RWr(6047)
//     PlcTask Inputs/PRG_MachineControl.fbMachineControler.fbRobot.fbCR800.stCR800EthercatData.arrRegistersInput[6048] <-> Module 1 (4 Stations:CR800 GPIO_REG_IF)/Tx PDO (4 Sta.)/RWr(6048)
//     PlcTask Inputs/PRG_MachineControl.fbMachineControler.fbRobot.fbCR800.stCR800EthercatData.arrRegistersInput[6049] <-> Module 1 (4 Stations:CR800 GPIO_REG_IF)/Tx PDO (4 Sta.)/RWr(6049)
//     PlcTask Inputs/PRG_MachineControl.fbMachineControler.fbRobot.fbCR800.stCR800EthercatData.arrRegistersInput[6050] <-> Module 1 (4 Stations:CR800 GPIO_REG_IF)/Tx PDO (4 Sta.)/RWr(6050)
//     PlcTask Inputs/PRG_MachineControl.fbMachineControler.fbRobot.fbCR800.stCR800EthercatData.arrRegistersInput[6051] <-> Module 1 (4 Stations:CR800 GPIO_REG_IF)/Tx PDO (4 Sta.)/RWr(6051)
//     PlcTask Inputs/PRG_MachineControl.fbMachineControler.fbRobot.fbCR800.stCR800EthercatData.arrRegistersInput[6052] <-> Module 1 (4 Stations:CR800 GPIO_REG_IF)/Tx PDO (4 Sta.)/RWr(6052)
//     PlcTask Inputs/PRG_MachineControl.fbMachineControler.fbRobot.fbCR800.stCR800EthercatData.arrRegistersInput[6053] <-> Module 1 (4 Stations:CR800 GPIO_REG_IF)/Tx PDO (4 Sta.)/RWr(6053)
//     PlcTask Inputs/PRG_MachineControl.fbMachineControler.fbRobot.fbCR800.stCR800EthercatData.arrRegistersInput[6054] <-> Module 1 (4 Stations:CR800 GPIO_REG_IF)/Tx PDO (4 Sta.)/RWr(6054)
//     PlcTask Inputs/PRG_MachineControl.fbMachineControler.fbRobot.fbCR800.stCR800EthercatData.arrRegistersInput[6055] <-> Module 1 (4 Stations:CR800 GPIO_REG_IF)/Tx PDO (4 Sta.)/RWr(6055)
//     PlcTask Inputs/PRG_MachineControl.fbMachineControler.fbRobot.fbCR800.stCR800EthercatData.arrRegistersInput[6056] <-> Module 1 (4 Stations:CR800 GPIO_REG_IF)/Tx PDO (4 Sta.)/RWr(6056)
//     PlcTask Inputs/PRG_MachineControl.fbMachineControler.fbRobot.fbCR800.stCR800EthercatData.arrRegistersInput[6057] <-> Module 1 (4 Stations:CR800 GPIO_REG_IF)/Tx PDO (4 Sta.)/RWr(6057)
//     PlcTask Inputs/PRG_MachineControl.fbMachineControler.fbRobot.fbCR800.stCR800EthercatData.arrRegistersInput[6058] <-> Module 1 (4 Stations:CR800 GPIO_REG_IF)/Tx PDO (4 Sta.)/RWr(6058)
//     PlcTask Inputs/PRG_MachineControl.fbMachineControler.fbRobot.fbCR800.stCR800EthercatData.arrRegistersInput[6059] <-> Module 1 (4 Stations:CR800 GPIO_REG_IF)/Tx PDO (4 Sta.)/RWr(6059)
//     PlcTask Inputs/PRG_MachineControl.fbMachineControler.fbRobot.fbCR800.stCR800EthercatData.arrRegistersInput[6060] <-> Module 1 (4 Stations:CR800 GPIO_REG_IF)/Tx PDO (4 Sta.)/RWr(6060)
//     PlcTask Inputs/PRG_MachineControl.fbMachineControler.fbRobot.fbCR800.stCR800EthercatData.arrRegistersInput[6061] <-> Module 1 (4 Stations:CR800 GPIO_REG_IF)/Tx PDO (4 Sta.)/RWr(6061)
//     PlcTask Inputs/PRG_MachineControl.fbMachineControler.fbRobot.fbCR800.stCR800EthercatData.arrRegistersInput[6062] <-> Module 1 (4 Stations:CR800 GPIO_REG_IF)/Tx PDO (4 Sta.)/RWr(6062)
//     PlcTask Inputs/PRG_MachineControl.fbMachineControler.fbRobot.fbCR800.stCR800EthercatData.arrRegistersInput[6063] <-> Module 1 (4 Stations:CR800 GPIO_REG_IF)/Tx PDO (4 Sta.)/RWr(6063)
//     PlcTask Inputs/PRG_MachineControl.fbMachineControler.fbRobot.fbCR800.stCR800EthercatData.arrRegistersInput[6064] <-> Module 1 (4 Stations:CR800 GPIO_REG_IF)/Tx PDO (4 Sta.)/RWr(6064)
//     PlcTask Inputs/PRG_MachineControl.fbMachineControler.fbRobot.fbCR800.stCR800EthercatData.arrRegistersInput[6065] <-> Module 1 (4 Stations:CR800 GPIO_REG_IF)/Tx PDO (4 Sta.)/RWr(6065)
//     PlcTask Inputs/PRG_MachineControl.fbMachineControler.fbRobot.fbCR800.stCR800EthercatData.arrRegistersInput[6066] <-> Module 1 (4 Stations:CR800 GPIO_REG_IF)/Tx PDO (4 Sta.)/RWr(6066)
//     PlcTask Inputs/PRG_MachineControl.fbMachineControler.fbRobot.fbCR800.stCR800EthercatData.arrRegistersInput[6067] <-> Module 1 (4 Stations:CR800 GPIO_REG_IF)/Tx PDO (4 Sta.)/RWr(6067)
//     PlcTask Inputs/PRG_MachineControl.fbMachineControler.fbRobot.fbCR800.stCR800EthercatData.arrRegistersInput[6068] <-> Module 1 (4 Stations:CR800 GPIO_REG_IF)/Tx PDO (4 Sta.)/RWr(6068)
//     PlcTask Inputs/PRG_MachineControl.fbMachineControler.fbRobot.fbCR800.stCR800EthercatData.arrRegistersInput[6069] <-> Module 1 (4 Stations:CR800 GPIO_REG_IF)/Tx PDO (4 Sta.)/RWr(6069)
//     PlcTask Inputs/PRG_MachineControl.fbMachineControler.fbRobot.fbCR800.stCR800EthercatData.arrRegistersInput[6070] <-> Module 1 (4 Stations:CR800 GPIO_REG_IF)/Tx PDO (4 Sta.)/RWr(6070)
//     PlcTask Inputs/PRG_MachineControl.fbMachineControler.fbRobot.fbCR800.stCR800EthercatData.arrRegistersInput[6071] <-> Module 1 (4 Stations:CR800 GPIO_REG_IF)/Tx PDO (4 Sta.)/RWr(6071)
//     PlcTask Inputs/PRG_MachineControl.fbMachineControler.fbRobot.fbCR800.stCR800EthercatData.arrRegistersInput[6072] <-> Module 1 (4 Stations:CR800 GPIO_REG_IF)/Tx PDO (4 Sta.)/RWr(6072)
//     PlcTask Inputs/PRG_MachineControl.fbMachineControler.fbRobot.fbCR800.stCR800EthercatData.arrRegistersInput[6075] <-> Module 1 (4 Stations:CR800 GPIO_REG_IF)/Tx PDO (4 Sta.)/RWr(6075)
//     PlcTask Inputs/PRG_MachineControl.fbMachineControler.fbRobot.fbCR800.stCR800EthercatData.arrRegistersInput[6076] <-> Module 1 (4 Stations:CR800 GPIO_REG_IF)/Tx PDO (4 Sta.)/RWr(6076)
//     PlcTask Inputs/PRG_MachineControl.fbMachineControler.fbRobot.fbCR800.stCR800EthercatData.arrRegistersInput[6077] <-> Module 1 (4 Stations:CR800 GPIO_REG_IF)/Tx PDO (4 Sta.)/RWr(6077)
//     PlcTask Inputs/PRG_MachineControl.fbMachineControler.fbRobot.fbCR800.stCR800EthercatData.arrRegistersInput[6078] <-> Module 1 (4 Stations:CR800 GPIO_REG_IF)/Tx PDO (4 Sta.)/RWr(6078)
//     PlcTask Inputs/PRG_MachineControl.fbMachineControler.fbRobot.fbCR800.stCR800EthercatData.arrRegistersInput[6079] <-> Module 1 (4 Stations:CR800 GPIO_REG_IF)/Tx PDO (4 Sta.)/RWr(6079)
//     PlcTask Inputs/PRG_MachineControl.fbMachineControler.fbRobot.fbCR800.stCR800EthercatData.arrRegistersInput[6080] <-> Module 1 (4 Stations:CR800 GPIO_REG_IF)/Tx PDO (4 Sta.)/RWr(6080)
//     PlcTask Inputs/PRG_MachineControl.fbMachineControler.fbRobot.fbCR800.stCR800EthercatData.arrRegistersInput[6081] <-> Module 1 (4 Stations:CR800 GPIO_REG_IF)/Tx PDO (4 Sta.)/RWr(6081)
//     PlcTask Inputs/PRG_MachineControl.fbMachineControler.fbRobot.fbCR800.stCR800EthercatData.arrRegistersInput[6082] <-> Module 1 (4 Stations:CR800 GPIO_REG_IF)/Tx PDO (4 Sta.)/RWr(6082)
//     PlcTask Inputs/PRG_MachineControl.fbMachineControler.fbRobot.fbCR800.stCR800EthercatData.arrRegistersInput[6083] <-> Module 1 (4 Stations:CR800 GPIO_REG_IF)/Tx PDO (4 Sta.)/RWr(6083)
//     PlcTask Inputs/PRG_MachineControl.fbMachineControler.fbRobot.fbCR800.stCR800EthercatData.arrRegistersInput[6084] <-> Module 1 (4 Stations:CR800 GPIO_REG_IF)/Tx PDO (4 Sta.)/RWr(6084)
//     PlcTask Inputs/PRG_MachineControl.fbMachineControler.fbRobot.fbCR800.stCR800EthercatData.arrRegistersInput[6085] <-> Module 1 (4 Stations:CR800 GPIO_REG_IF)/Tx PDO (4 Sta.)/RWr(6085)
//     PlcTask Inputs/PRG_MachineControl.fbMachineControler.fbRobot.fbCR800.stCR800EthercatData.arrRegistersInput[6086] <-> Module 1 (4 Stations:CR800 GPIO_REG_IF)/Tx PDO (4 Sta.)/RWr(6086)
//     PlcTask Inputs/PRG_MachineControl.fbMachineControler.fbRobot.fbCR800.stCR800EthercatData.arrRegistersInput[6087] <-> Module 1 (4 Stations:CR800 GPIO_REG_IF)/Tx PDO (4 Sta.)/RWr(6087)
//     PlcTask Inputs/PRG_MachineControl.fbMachineControler.fbRobot.fbCR800.stCR800EthercatData.arrRegistersInput[6088] <-> Module 1 (4 Stations:CR800 GPIO_REG_IF)/Tx PDO (4 Sta.)/RWr(6088)
//     PlcTask Inputs/PRG_MachineControl.fbMachineControler.fbRobot.fbCR800.stCR800EthercatData.arrRegistersInput[6089] <-> Module 1 (4 Stations:CR800 GPIO_REG_IF)/Tx PDO (4 Sta.)/RWr(6089)
//     PlcTask Inputs/PRG_MachineControl.fbMachineControler.fbRobot.fbCR800.stCR800EthercatData.arrRegistersInput[6090] <-> Module 1 (4 Stations:CR800 GPIO_REG_IF)/Tx PDO (4 Sta.)/RWr(6090)
//     PlcTask Inputs/PRG_MachineControl.fbMachineControler.fbRobot.fbCR800.stCR800EthercatData.arrRegistersInput[6091] <-> Module 1 (4 Stations:CR800 GPIO_REG_IF)/Tx PDO (4 Sta.)/RWr(6091)
//     PlcTask Inputs/PRG_MachineControl.fbMachineControler.fbRobot.fbCR800.stCR800EthercatData.arrRegistersInput[6092] <-> Module 1 (4 Stations:CR800 GPIO_REG_IF)/Tx PDO (4 Sta.)/RWr(6092)
//     PlcTask Inputs/PRG_MachineControl.fbMachineControler.fbRobot.fbCR800.stCR800EthercatData.arrRegistersInput[6093] <-> Module 1 (4 Stations:CR800 GPIO_REG_IF)/Tx PDO (4 Sta.)/RWr(6093)
//     PlcTask Inputs/PRG_MachineControl.fbMachineControler.fbRobot.fbCR800.stCR800EthercatData.arrRegistersInput[6094] <-> Module 1 (4 Stations:CR800 GPIO_REG_IF)/Tx PDO (4 Sta.)/RWr(6094)
//     PlcTask Inputs/PRG_MachineControl.fbMachineControler.fbRobot.fbCR800.stCR800EthercatData.arrRegistersInput[6095] <-> Module 1 (4 Stations:CR800 GPIO_REG_IF)/Tx PDO (4 Sta.)/RWr(6095)
//     PlcTask Inputs/PRG_MachineControl.fbMachineControler.fbRobot.fbCR800.stCR800EthercatData.arrRegistersInput[6096] <-> Module 1 (4 Stations:CR800 GPIO_REG_IF)/Tx PDO (4 Sta.)/RWr(6096)
//     PlcTask Inputs/PRG_MachineControl.fbMachineControler.fbRobot.fbCR800.stCR800EthercatData.arrRegistersInput[6097] <-> Module 1 (4 Stations:CR800 GPIO_REG_IF)/Tx PDO (4 Sta.)/RWr(6097)
//     PlcTask Inputs/PRG_MachineControl.fbMachineControler.fbRobot.fbCR800.stCR800EthercatData.arrRegistersInput[6098] <-> Module 1 (4 Stations:CR800 GPIO_REG_IF)/Tx PDO (4 Sta.)/RWr(6098)
//     PlcTask Inputs/PRG_MachineControl.fbMachineControler.fbRobot.fbCR800.stCR800EthercatData.arrRegistersInput[6099] <-> Module 1 (4 Stations:CR800 GPIO_REG_IF)/Tx PDO (4 Sta.)/RWr(6099)
//     PlcTask Inputs/PRG_MachineControl.fbMachineControler.fbRobot.fbCR800.stCR800EthercatData.arrRegistersInput[6100] <-> Module 1 (4 Stations:CR800 GPIO_REG_IF)/Tx PDO (4 Sta.)/RWr(6100)
//     PlcTask Inputs/PRG_MachineControl.fbMachineControler.fbRobot.fbCR800.stCR800EthercatData.arrRegistersInput[6101] <-> Module 1 (4 Stations:CR800 GPIO_REG_IF)/Tx PDO (4 Sta.)/RWr(6101)
//     PlcTask Inputs/PRG_MachineControl.fbMachineControler.fbRobot.fbCR800.stCR800EthercatData.arrRegistersInput[6102] <-> Module 1 (4 Stations:CR800 GPIO_REG_IF)/Tx PDO (4 Sta.)/RWr(6102)
//     PlcTask Inputs/PRG_MachineControl.fbMachineControler.fbRobot.fbCR800.stCR800EthercatData.arrRegistersInput[6103] <-> Module 1 (4 Stations:CR800 GPIO_REG_IF)/Tx PDO (4 Sta.)/RWr(6103)
//     PlcTask Inputs/PRG_MachineControl.fbMachineControler.fbRobot.fbCR800.stCR800EthercatData.arrRegistersInput[6104] <-> Module 1 (4 Stations:CR800 GPIO_REG_IF)/Tx PDO (4 Sta.)/RWr(6104)
//     PlcTask Inputs/PRG_MachineControl.fbMachineControler.fbRobot.fbCR800.stCR800EthercatData.arrRegistersInput[6105] <-> Module 1 (4 Stations:CR800 GPIO_REG_IF)/Tx PDO (4 Sta.)/RWr(6105)
//     PlcTask Inputs/PRG_MachineControl.fbMachineControler.fbRobot.fbCR800.stCR800EthercatData.arrRegistersInput[6106] <-> Module 1 (4 Stations:CR800 GPIO_REG_IF)/Tx PDO (4 Sta.)/RWr(6106)
//     PlcTask Inputs/PRG_MachineControl.fbMachineControler.fbRobot.fbCR800.stCR800EthercatData.arrRegistersInput[6107] <-> Module 1 (4 Stations:CR800 GPIO_REG_IF)/Tx PDO (4 Sta.)/RWr(6107)
//     PlcTask Inputs/PRG_MachineControl.fbMachineControler.fbRobot.fbCR800.stCR800EthercatData.arrRegistersInput[6108] <-> Module 1 (4 Stations:CR800 GPIO_REG_IF)/Tx PDO (4 Sta.)/RWr(6108)
//     PlcTask Inputs/PRG_MachineControl.fbMachineControler.fbRobot.fbCR800.stCR800EthercatData.arrRegistersInput[6109] <-> Module 1 (4 Stations:CR800 GPIO_REG_IF)/Tx PDO (4 Sta.)/RWr(6109)
//     PlcTask Inputs/PRG_MachineControl.fbMachineControler.fbRobot.fbCR800.stCR800EthercatData.arrRegistersInput[6110] <-> Module 1 (4 Stations:CR800 GPIO_REG_IF)/Tx PDO (4 Sta.)/RWr(6110)
//     PlcTask Inputs/PRG_MachineControl.fbMachineControler.fbRobot.fbCR800.stCR800EthercatData.arrRegistersInput[6111] <-> Module 1 (4 Stations:CR800 GPIO_REG_IF)/Tx PDO (4 Sta.)/RWr(6111)
//     PlcTask Inputs/PRG_MachineControl.fbMachineControler.fbRobot.fbCR800.stCR800EthercatData.arrRegistersInput[6112] <-> Module 1 (4 Stations:CR800 GPIO_REG_IF)/Tx PDO (4 Sta.)/RWr(6112)
//     PlcTask Inputs/PRG_MachineControl.fbMachineControler.fbRobot.fbCR800.stCR800EthercatData.arrRegistersInput[6113] <-> Module 1 (4 Stations:CR800 GPIO_REG_IF)/Tx PDO (4 Sta.)/RWr(6113)
//     PlcTask Inputs/PRG_MachineControl.fbMachineControler.fbRobot.fbCR800.stCR800EthercatData.arrRegistersInput[6114] <-> Module 1 (4 Stations:CR800 GPIO_REG_IF)/Tx PDO (4 Sta.)/RWr(6114)
//     PlcTask Inputs/PRG_MachineControl.fbMachineControler.fbRobot.fbCR800.stCR800EthercatData.arrRegistersInput[6115] <-> Module 1 (4 Stations:CR800 GPIO_REG_IF)/Tx PDO (4 Sta.)/RWr(6115)
//     PlcTask Inputs/PRG_MachineControl.fbMachineControler.fbRobot.fbCR800.stCR800EthercatData.arrRegistersInput[6116] <-> Module 1 (4 Stations:CR800 GPIO_REG_IF)/Tx PDO (4 Sta.)/RWr(6116)
//     PlcTask Inputs/PRG_MachineControl.fbMachineControler.fbRobot.fbCR800.stCR800EthercatData.arrRegistersInput[6117] <-> Module 1 (4 Stations:CR800 GPIO_REG_IF)/Tx PDO (4 Sta.)/RWr(6117)
//     PlcTask Inputs/PRG_MachineControl.fbMachineControler.fbRobot.fbCR800.stCR800EthercatData.arrRegistersInput[6118] <-> Module 1 (4 Stations:CR800 GPIO_REG_IF)/Tx PDO (4 Sta.)/RWr(6118)
//     PlcTask Inputs/PRG_MachineControl.fbMachineControler.fbRobot.fbCR800.stCR800EthercatData.arrRegistersInput[6119] <-> Module 1 (4 Stations:CR800 GPIO_REG_IF)/Tx PDO (4 Sta.)/RWr(6119)
//     PlcTask Inputs/PRG_MachineControl.fbMachineControler.fbRobot.fbCR800.stCR800EthercatData.arrRegistersInput[6120] <-> Module 1 (4 Stations:CR800 GPIO_REG_IF)/Tx PDO (4 Sta.)/RWr(6120)
//     PlcTask Inputs/PRG_MachineControl.fbMachineControler.fbRobot.fbCR800.stCR800EthercatData.arrRegistersInput[6121] <-> Module 1 (4 Stations:CR800 GPIO_REG_IF)/Tx PDO (4 Sta.)/RWr(6121)
//     PlcTask Inputs/PRG_MachineControl.fbMachineControler.fbRobot.fbCR800.stCR800EthercatData.arrRegistersInput[6122] <-> Module 1 (4 Stations:CR800 GPIO_REG_IF)/Tx PDO (4 Sta.)/RWr(6122)
//     PlcTask Inputs/PRG_MachineControl.fbMachineControler.fbRobot.fbCR800.stCR800EthercatData.arrRegistersInput[6124] <-> Module 1 (4 Stations:CR800 GPIO_REG_IF)/Tx PDO (4 Sta.)/RWr(6124)
//     PlcTask Inputs/PRG_MachineControl.fbMachineControler.fbRobot.fbCR800.stCR800EthercatData.arrRegistersInput[6125] <-> Module 1 (4 Stations:CR800 GPIO_REG_IF)/Tx PDO (4 Sta.)/RWr(6125)
//     PlcTask Inputs/PRG_MachineControl.fbMachineControler.fbRobot.fbCR800.stCR800EthercatData.arrRegistersInput[6126] <-> Module 1 (4 Stations:CR800 GPIO_REG_IF)/Tx PDO (4 Sta.)/RWr(6126)
//     PlcTask Inputs/PRG_MachineControl.fbMachineControler.fbRobot.fbCR800.stCR800EthercatData.arrRegistersInput[6127] <-> Module 1 (4 Stations:CR800 GPIO_REG_IF)/Tx PDO (4 Sta.)/RWr(6127)
//     PlcTask Inputs/PRG_MachineControl.fbMachineControler.fbRobot.fbCR800.stCR800EthercatData.arrRegistersInput[6073] <-> Module 1 (4 Stations:CR800 GPIO_REG_IF)/Tx PDO (4 Sta.)/
RWr(6073)
//     PlcTask Inputs/PRG_MachineControl.fbMachineControler.fbRobot.fbCR800.stCR800EthercatData.arrRegistersInput[6074] <-> Module 1 (4 Stations:CR800 GPIO_REG_IF)/Tx PDO (4 Sta.)/
RWr(6074)
//     PlcTask Inputs/PRG_MachineControl.fbMachineControler.fbRobot.fbCR800.stCR800EthercatData.arrRegistersInput[6123] <-> Module 1 (4 Stations:CR800 GPIO_REG_IF)/Tx PDO (4 Sta.)/
RWr(6123)
//     PlcTask Inputs/PRG_MachineControl.fbMachineControler.fbRobot.fbCR800.stCR800EthercatData.arrSignalsInputRaw[{0..31}] <-> Module 1 (4 Stations:CR800 GPIO_REG_IF)/Tx PDO (4 Sta.)/RX({6000..6248 step 8}-{6007..6255 step 8})  (32 links)
//     PlcTask Inputs/PRG_MachineControl.fbMachineControler.fbRobot.fbCR800.stCR800EthercatData.iInfoDataState <-> InfoData/State
//     PlcTask Outputs/PRG_MachineControl.fbMachineControler.fbRobot.fbCR800.stCR800EthercatData.arrRegistersOutput[{6000..6127}] <-> Module 1 (4 Stations:CR800 GPIO_REG_IF)/Rx PDO (4 Sta.)/RWw({6000..6127})  (128 links)
//     PlcTask Outputs/PRG_MachineControl.fbMachineControler.fbRobot.fbCR800.stCR800EthercatData.arrSignalsOutputRaw[{0..31}] <-> Module 1 (4 Stations:CR800 GPIO_REG_IF)/Rx PDO (4 Sta.)/RY({6000..6248 step 8}-{6007..6255 step 8})  (32 links)
//   PShEll_UniversalBlocks/PShEll_UniversalBlocks Instance <-> Device 1 (EtherCAT)/Term 1 (EK1200)/Term 20 (EK1122)/Box 23 (EX260-SEC1)
//     PlcTask Outputs/PRG_MachineControl.fbMachineControler.doBlowBowlFeeder.bOut <-> Byte 0/Output
//     PlcTask Outputs/PRG_MachineControl.fbMachineControler.doBlowDentContamination.bOut <-> Byte 0/Output @bit 4
//     PlcTask Outputs/PRG_MachineControl.fbMachineControler.doBlowDirtScratch.bOut <-> Byte 0/Output @bit 6
//     PlcTask Outputs/PRG_MachineControl.fbMachineControler.doBlowGood.bOut <-> Byte 0/Output @bit 2
//     PlcTask Outputs/PRG_MachineControl.fbMachineControler.doBlowReject.bOut <-> Byte 1/Output
//   PShEll_UniversalBlocks/PShEll_UniversalBlocks Instance <-> Device 1 (EtherCAT)/Term 1 (EK1200)/Term 5 (EL1114)
//     PlcTask Inputs/PRG_MachineControl.fbMachineControler.diProductPresenceBowl.bIn <-> Channel 3/Input
//   PShEll_UniversalBlocks/PShEll_UniversalBlocks Instance <-> Device 1 (EtherCAT)/Term 1 (EK1200)/Term 7 (EL2004)
//     PlcTask Outputs/PRG_MachineControl.fbMachineControler.poDoorLock.bOut <-> Channel 2/Output
//     PlcTask Outputs/PRG_MachineControl.fbMachineControler.poResetButtonLight.bOut <-> Channel 1/Output
//   PShEll_UniversalBlocks/PShEll_UniversalBlocks Instance <-> Device 1 (EtherCAT)/Term 1 (EK1200)/Term 9 (EL1114)
//     PlcTask Inputs/PRG_MachineControl.fbMachineControler.fbRotaryTable.piHomeSwitch.bIn <-> Channel 4/Input
//   PShEll_UniversalBlocks/PShEll_UniversalBlocks Instance <-> NC-Task 1 SAF/Axes/Rotary Table
//     PlcTask Inputs/PRG_MachineControl.fbMachineControler.fbRotaryTable.stAxisRef.NcToPlc <-> Outputs/ToPlc
//     PlcTask Outputs/PRG_MachineControl.fbMachineControler.fbRotaryTable.stAxisRef.PlcToNc <-> Inputs/FromPlc

CONFIGURATION PShEll_UniversalBlocks
    RESOURCE PLC ON TwinCAT3
        TASK PlcTask(INTERVAL := T#10ms, PRIORITY := 20);
        TASK VISU_TASK(INTERVAL := T#100000us, PRIORITY := 30);
        PROGRAM PRG_VisuControl WITH PlcTask : PRG_VisuControl;
        PROGRAM PRG_AlarmControl WITH PlcTask : PRG_AlarmControl;
        PROGRAM PRG_MachineControl WITH PlcTask : PRG_MachineControl;
        PROGRAM PRG_RecipesManager WITH PlcTask : PRG_RecipesManager;
        PROGRAM VisuElems_Visu_Prg WITH VISU_TASK : VisuElems.Visu_Prg;
    END_RESOURCE
END_CONFIGURATION

// ---- DUTs/Libs/BowlFeeder/E_BowlFeederUnitState.TcDUT
{attribute 'strict'}
TYPE E_BowlFeederUnitState :
(
	BOWL_FEEDER_UNIT_UNINITIALIZED 		:= 0,
	BOWL_FEEDER_UNIT_INITIALIZING 		:= 10,
	BOWL_FEEDER_UNIT_READY_INITIALIZED 	:= 20,
	
	BOWL_FEEDER_UNIT_IDLE 				:= 30,		(* Ready to work *)
	BOWL_FEEDER_UNIT_START				:= 40,
	BOWL_FEEDER_UNIT_RUNNING			:= 50,
	BOWL_FEEDER_UNIT_STOP				:= 60,
	BOWL_FEEDER_UNIT_STOP_DONE			:= 70,
	
	BOWL_FEEDER_UNIT_ABORT				:= 80
);	
END_TYPE

// ---- DUTs/Libs/BowlFeeder/E_BowlFeederUnitStateInit.TcDUT
{attribute 'strict'}
TYPE E_BowlFeederUnitStateInit :
(
	BOWL_FEEDER_UNIT_INIT_START 		:= 0,
	BOWL_FEEDER_UNIT_INIT_RUNNING_CHECK := 10,
	BOWL_FEEDER_UNIT_INIT_STOP 			:= 20,
	BOWL_FEEDER_UNIT_INIT_STOP_CHECK	:= 30,
	BOWL_FEEDER_UNIT_INIT_DONE 			:= 40
);
END_TYPE

// ---- DUTs/Libs/Platform/Universal Visu/E_VisuCtrlPageState.TcDUT
{attribute 'strict'}
TYPE E_VisuCtrlPageState :
(
	SCREEN_UNINITIALIZED 		:= 0,	(*  *)
	SCREEN_INITIALIZING 		:= 1,	(*  *)
	SCREEN_READY_INITIALIZED	:= 2,	(*  *)
	SCREEN_AUTO					:= 3,	(*  *)
	SCREEN_MODE_CHANGE			:= 4,	(*  *)
	SCREEN_MANUAL_CYLINDERS		:= 9,	(*  *)
	SCREEN_MANUAL_MOTORS		:= 8,	(*  *)
	//SCREEN_MANUAL_SAFETY		:= 7,	(*  *)
	SCREEN_MANUAL_INPUTS		:= 11,	(*  *)
	SCREEN_MANUAL_OUTPUTS		:= 16,	(*  *)
	SCREEN_MANUAL_ROBOTS		:= 5,	(*  *)
	SCREEN_MANUAL_OTHERS		:= 10,	(*  *)
	SCREEN_ALARMS				:= 7,	(*  *)
	SCREEN_RECIPES				:= 12,	(*  *)
	SCREEN_RESET				:= 13,	(*  *)
	SCREEN_ABORTING				:= 6,	(*  *)
	SCREEN_EMERGENCY			:= 15	(*  *)
);
END_TYPE

// ---- DUTs/Libs/Platform/Universal Visu/ST_VisuCtrlCylinderFrame.TcDUT
TYPE ST_VisuCtrlCylinderFrame EXTENDS ST_VisuCtrlUnitFrame :
STRUCT
	btnInit				: BOOL;				(*  *)
	btnAbort			: BOOL;				(*  *)
	btnReset			: BOOL;				(*  *)
	btnGoHome 			: BOOL;				(*  *)
	btnGoActive 		: BOOL;				(*  *)
	btnRealase 			: BOOL;				(*  *)
	
	bSensorHome 		: BOOL;				(*  *)
	bSensorActive 		: BOOL;				(*  *)
	bPositionHold		: BOOL;				(*  *)
	bError				: BOOL;				(*  *)
	iErrorID			: INT;				(*  *)
	
	tActiveMovement 	: TIME;				(*  *)
	tHomeMovement 		: TIME;				(*  *)
	
	sActiveDescription 	: STRING;			(*  *)
	sHomeDescription 	: STRING;			(*  *)
	sStateDescription	: STRING;			(*  *)
	
	sCylinderImage		: STRING;			(*  *)
	eCylinderState		: E_CylinderState;	(*  *)
END_STRUCT
END_TYPE

// ---- DUTs/Libs/SMC SI Unit/ST_EX260_SEC1.TcDUT
TYPE ST_EX260_SEC1 :
STRUCT
	arrSignalsOutputRaw			AT%Q*	: ARRAY[0..3] 		OF BYTE ; 		(*Output process data (RX) before convertion to easier to use. 
																			This data are is used only in MR_ConvertEthercatData*)
	arrSignalsOutputConverted			: ARRAY[1..32] OF BOOL ; 		(*Output process data (RX) after convertion to esier to uses. 
																			  This data are used in program*)
END_STRUCT
END_TYPE

// ---- DUTs/Machine/Machine Control/Batch/ST_BatchData.TcDUT
TYPE ST_BatchData :
STRUCT
	sBatchID			: STRING;
	sProductionOrder 	: STRING;
	sOperatorID			: STRING;
	sProductItemConfig	: STRING;
	sInputQuantity		: STRING;
END_STRUCT
END_TYPE

// ---- DUTs/Machine/Machine Control/Batch/ST_BatchPerformacne.TcDUT
TYPE ST_BatchPerformacne :
STRUCT
	iBatchProgress							: USINT;

	iCurrentQuantity						: USINT;
	iGoodQuantity 							: USINT;
	iReworkQuantity							: USINT;
	iReworkDirtyQuantity					: USINT;
	iReworkDentQuantity						: USINT;
	iRejectedQuantity						: USINT;

	iRejectLessQttyCamQuantity				: USINT;
	iRejectLessQttyHoleQuantity				: USINT;
	iRejectLessQttySoundOutletQuantity		: USINT;
	iRejectStoneStuckInHoleQuantity			: USINT;
	iRejectContaminationQuantity			: USINT;
	iRejectDeformQuantity					: USINT;
	iRejectInsufficienctQuantity			: USINT;
	iRejectBurrQuantity						: USINT;
	iRejectScratchQuantity					: USINT;
	iRejectDentQuantity						: USINT;

	bMachineStart							: BOOL;
	bMachineStop							: BOOL;
END_STRUCT
END_TYPE

// ---- DUTs/Machine/Machine Control/E_MachineCtrlStateAbort.TcDUT
{attribute 'strict'}
TYPE E_MachineCtrlStateAbort :
(
	MACHINE_STATE_ABORTING_TABLE					:= 0,	(*  *)
	MACHINE_STATE_ABORTING_ROBOT_CYCLE_STOP			:= 10,	(*  *)
	MACHINE_STATE_ABORTING_DONE						:= 200	(*  *)
);
END_TYPE

// ---- DUTs/Machine/Machine Control/E_MachineCtrlStateAuto.TcDUT
{attribute 'strict'}
TYPE E_MachineCtrlStateAuto :
(
	MACHINE_STATE_AUTO_IDLE 	:= 0,
	MACHINE_STATE_AUTO_RUNNING 	:= 10
);
END_TYPE

// ---- DUTs/Machine/Machine Control/E_MachineCtrlStateAutoAOI.TcDUT
{attribute 'strict'}
TYPE E_MachineCtrlStateAutoAOI :
(
	MACHINE_STATE_AUTO_AOI_IDLE 				:= 0,	(* During this state machine is waiting for choosing one of workmode and additional parameters *)
	MACHINE_STATE_AUTO_AOI_PROCCESSING		:= 10,
	MACHINE_STATE_AUTO_AOI_GO_INPUT				:= 20,
	MACHINE_STATE_AUTO_AOI_GO_BACK				:= 30,		
	MACHINE_STATE_AUTO_AOI_DONE					:= 40
)UINT;
END_TYPE

// ---- DUTs/Machine/Machine Control/E_MachineCtrlStateInit.TcDUT
{attribute 'strict'}
TYPE E_MachineCtrlStateInit :
(	
	(* Safety init *)
	MACHINE_STATE_INITIALIZING_MACHINE_LOGGER					:= 0,	(*  *)
	MACHINE_STATE_INITIALIZING_RECIPES_MANAGER					:= 10,	(*  *)
	MACHINE_STATE_INITIALIZING_CLEAR_ALL_ERRORS					:= 20,	(*  *)
	MACHINE_STATE_INITIALIZING_SAFETY_INITIALIZATION			:= 50,	(*  *)
	MACHINE_STATE_INITIALIZING_CHECK_ESTOP						:= 60,	(*  *)
	MACHINE_STATE_INITIALIZING_CHECK_DOOR_LOCKS					:= 80,	(*  *)
	MACHINE_STATE_INITIALIZING_ROBOTS_POWER_CHECK				:= 90,	(*  *)
	MACHINE_STATE_INITIALIZING_SAFETY_RESET						:= 100,	(*  *)
	MACHINE_STATE_INITIALIZING_SAFETY_START						:= 110,	(*  *)
	MACHINE_STATE_INITIALIZING_ROBOT_CONTROLERS_RESET			:= 120,	(*  *)
	MACHINE_STATE_INITIALIZING_SAFETY_CHECK						:= 130,	(*  *)
	MACHINE_STATE_INITIALIZING_ROBOT_AUTO_MODE_SW				:= 140,
	
	(* Robot init *)                                          		
	MACHINE_STATE_INITIALIZING_ROBOT_ABORT						:= 200,	(*  *)
	MACHINE_STATE_INITIALIZING_ROBOT_INIT						:= 210,	(*  *)
	MACHINE_STATE_INITIALIZING_ROBOT_HOME						:= 220,	(*  *)
	MACHINE_STATE_INITIALIZING_ROBOT_AUTOMATIC_MODE				:= 230,	(*  *)
	
	(* Rotary table init *)
	MACHINE_STATE_INITIALIZING_ROTARY_TABLE_ABORT				:= 400,
	MACHINE_STATE_INITIALIZING_ROTARY_TABLE_INIT				:= 410,	(*  *)
	MACHINE_STATE_INITIALIZING_ROTARY_TABLE_HOME				:= 420,	(*  *)

	(* Bowl feeder init *)
	MACHINE_STATE_INITIALIZING_BOWL_INIT						:= 500,
	
	(* RTC Vision System init *)
	MACHINE_STATE_INITIALIZING_RTC_VISION_INIT					:= 600,

	MACHINE_STATE_INITIALIZING_DONE								:= 1000	(*  *)
)UINT;
END_TYPE

// ---- DUTs/Machine/Machine Control/E_MachineCtrlStateManualToAuto.TcDUT
{attribute 'strict'}
TYPE E_MachineCtrlStateManualToAuto :
(
	
	MACHINE_STATE_MANUAL_TO_AUTO_ROBOT_CYCLE_STOP			:= 0,	(*  *)

	MACHINE_STATE_MANUAL_TO_AUTO_ROBOT_ABORT				:= 10,	(*  *)
	MACHINE_STATE_MANUAL_TO_AUTO_ROBOT_REMOTE_MODE			:= 20,	(*  *)
	MACHINE_STATE_MANUAL_TO_AUTO_ROBOT_INIT					:= 30,	(*  *)
	MACHINE_STATE_MANUAL_TO_AUTO_ROBOT_HOME					:= 40,	(*  *)
	MACHINE_STATE_MANUAL_TO_AUTO_ROBOT_AUTOMATIC_MODE		:= 50,	(*  *)
                 
	MACHINE_STATE_MANUAL_TO_AUTO_DONE						:= 260
);
END_TYPE

// ---- DUTs/Machine/Machine Control/E_MachineCtrlStateUninitialized.TcDUT
{attribute 'strict'}
TYPE E_MachineCtrlStateUninitialized :
(	
	(*Robot uninitializing *)
	MACHINE_STATE_UNINITIALIZED_POWER_ON_CR800 						:= 0,	
	MACHINE_STATE_UNINITIALIZED_CR800_ETHERCAT_STATUS_CHECK 		:= 10,
	MACHINE_STATE_UNINITIALIZED_CR800_ETHERCAT_STATUS_CHECK_DONE	:= 20,
	MACHINE_STATE_UNINITIALIZED_CR800_ETHERCAT_ERROR_RESET			:= 30,
	MACHINE_STATE_UNINITIALIZED_CR800_ETHERCAT_REQUEST_OP_STATE		:= 40,	(*  *)	
	MACHINE_STATE_UNINITIALIZED_CR800_CHECK_POWER_REGISTER			:= 50,	(*  *)
	
	MACHINE_STATE_UNINITIALIZED_DONE								:= 60	(*  *)
);
END_TYPE

// ---- DUTs/Machine/Machine Control/Internal/E_GoldenSampleMeasurementState.TcDUT
{attribute 'strict'}
TYPE E_GoldenSampleMeasurementState :
(
	GOLDEN_SAMPLE_MEASUREMENT_IDLE 									:= 0,
	
	GOLDEN_SAMPLE_MEASUREMENT_ROBOT_GO_TO_SAMPLE					:= 40,
	GOLDEN_SAMPLE_MEASUREMENT_ROBOT_PICK_SAMPLE						:= 50,
	
	GOLDEN_SAMPLE_MEASUREMENT_ROBOT_GO_TO_STATION_1					:= 60,
	GOLDEN_SAMPLE_MEASUREMENT_ROBOT_GO_TO_STATION_1_DONE			:= 70,
	GOLDEN_SAMPLE_MEASUREMENT_ROBOT_GO_TO_STATION_2					:= 80,
	GOLDEN_SAMPLE_MEASUREMENT_ROBOT_GO_TO_STATION_2_DONE			:= 90,
	
	GOLDEN_SAMPLE_MEASUREMENT_ROBOT_GO_TO_REJECTBOX					:= 100,
	GOLDEN_SAMPLE_MEASUREMENT_ROBOT_GO_TO_ROTARY_TABLE				:= 110,
	GOLDEN_SAMPLE_MEASUREMENT_ROBOT_DROP_PRODUCT_ROTARY_TABLE		:= 115,
	GOLDEN_SAMPLE_MEASUREMENT_ROBOT_DROP_PRODUCT_ROTARY_TABLE_DONE	:= 120,
	
	GOLDEN_SAMPLE_MEASUREMENT_ROBOT_GO_TO_OUT_POSITION				:= 130,
	GOLDEN_SAMPLE_MEASUREMENT_ROBOT_GO_TO_OUT_POSITION_PICK			:= 135,
		
	GOLDEN_SAMPLE_MEASUREMENT_ROBOT_RETURN_TO_STATION				:= 140,
	GOLDEN_SAMPLE_MEASUREMENT_ROBOT_RETURN_TO_STATION_PLACED		:= 150,
	GOLDEN_SAMPLE_MEASUREMENT_ROBOT_RETURN_TO_STATION_PLACED_DONE	:= 160,
	
	GOLDEN_SAMPLE_MEASUREMENT_CHECK_RESULTS							:= 180,
	
	GOLDEN_SAMPLE_MEASUREMENT_GO_SAFE_POSITION						:= 190,
	GOLDEN_SAMPLE_MEASUREMENT_SAFE_POSITION_DONE					:= 200,
	
	GOLDEN_SAMPLE_MEASUREMENT_OK 									:= 210,
	GOLDEN_SAMPLE_MEASUREMENT_FAIL 									:= 220,
	GOLDEN_SAMPLE_MEASUREMENT_STOPPED								:= 230
);
END_TYPE

// ---- DUTs/Machine/Machine Control/Internal/E_RotaryTableState.TcDUT
{attribute 'strict'}
TYPE E_RotaryTableState :
(
	ROTARY_TABLE_IDLE 					:= 0,	(*  *)
	ROTARY_TABLE_ROBOT_IN_POSITION 		:= 10,	(*  *)
	ROTARY_TABLE_ROBOT_DROP_PRODUCT		:= 20,	(*  *)
	ROTARY_TABLE_MOVE_TO_STATION_1		:= 30,	(*  *)
	ROTARY_TABLE_SEND_COMMAND_STATION1	:= 40	(*  *)
	
);
END_TYPE

// ---- DUTs/Machine/Shell API/ST_ShellPlatform.TcDUT
TYPE ST_ShellPlatform EXTENDS ST_UniversalPlatform :
STRUCT
	ref_fbMachineControler : REFERENCE TO FB_MachineControl;	(*  *)
	ref_MachineSafety	: REFERENCE TO FB_MachineSafety;	(*  *)
	ref_fbVisuControler	: REFERENCE TO FB_VisuControl;			(*  *)
END_STRUCT
END_TYPE

// ---- DUTs/Machine/Visu Control/E_VisuCtrlInitializingPopUpFrameSelector.TcDUT
{attribute 'strict'}
TYPE E_VisuCtrlInitializingPopUpFrameSelector :
(
	VISU_CTRL_INITIALIZING_FRAME_E_STOP 					:= 0,
	VISU_CTRL_INITIALIZING_FRAME_DOOR_LOCK 					:= 1,	
	VISU_CTRL_INITIALIZING_FRAME_RESET_BUTTON				:= 3	
);
END_TYPE

// ---- DUTs/Machine/Visu Control/E_VisuCtrlUninitializedFrameSelector.TcDUT
{attribute 'strict'}
TYPE E_VisuCtrlUninitializedFrameSelector :
(
	VISU_CTRL_UNINITIALIZED_FRAME_STARTUP 	:= 0,
	VISU_CTRL_UNINITIALIZED_FRAME_SETUP		:= 1
);
END_TYPE

// ---- DUTs/Machine/Visu Control/ST_InitializationFrame.TcDUT
TYPE ST_InitializationFrame :
STRUCT
	bMachineLoggerInitialized	: BOOL;												(* Platform machine logger initialized*)
	bRecipesManagerInitialized	: BOOL;												(* Platform recipes manager initialized *)
	bMesConnected 				: BOOL;												(* Machine connected to the MES *)
	bSafetyInitialization		: BOOL;												(*  *)
	bEStopChecked				: BOOL;												(*  *)
	bCourtainChecked			: BOOL;												(*  *)
	bDoorsLocked				: BOOL;												(* Machine door's locked *)
	bRobotControlersPowerOn		: BOOL;												(* Robots controlers power on *)
	bSafetyReset				: BOOL;												(* Safety status checked *)
	bSafetyStart				: BOOL;												(* Safety started *) 
	bRobotControlersResetDone	: BOOL;												(* Robots controlers reset done *)
	bSafetyCheck				: BOOL;												(* Safety final status OK *)
	bRobotsInRemoteMode			: BOOL;												(* Robot controlers in remote mode *)
	bRobotOneInitialized 		: BOOL;												(* Robot one initialized *)
	bRobotTwoInitialized 		: BOOL;												(* Robot two initialized *)
	bRobotOneHomed				: BOOL;												(* Robot one homed *)
	bRobotTwoHomed				: BOOL;												(* Robot two homed *)
	bRobotsInAutomaticMode		: BOOL;												(*  *)
	
END_STRUCT
END_TYPE

// ---- DUTs/Machine/Visu Control/ST_UninitializedSetupFrame.TcDUT
TYPE ST_UninitializedSetupFrame :
STRUCT
	(* --- Communication setup --- *)
	(* MES *)
	sMesIpAddress 				: T_IPv4Addr;					(*  *)
	iMesPort					: UINT;							(*  *)
	
	(* Camera *)
	sCameraIpAddress			: T_IPv4Addr;					(*  *)
	iCameraPort					: UINT;							(*  *)
	
END_STRUCT
END_TYPE

// ---- DUTs/Machine/Visu Control/ST_UninitializedStartUpFrame.TcDUT
TYPE ST_UninitializedStartUpFrame :
STRUCT
	iProgressBar					: USINT;
	bRTCVisionPowerOn				: BOOL;
	bCR800PowerOn					: BOOL;
	bCR800EtherCatInitialization	: BOOL;
END_STRUCT
END_TYPE

// ---- POUs/Machine/Module/Robot/E_AOIRobotActions.TcDUT
{attribute 'strict'}
TYPE E_AOIRobotActions :
(
	AOI_ROBOT_ACTION_PICK					:= 60,
	AOI_ROBOT_ACTION_PLACE					:= 61,
	AOI_ROBOT_ACTION_GO_BOWL				:= 62,	
	AOI_ROBOT_ACTION_GO_TO_STATION_1		:= 63,
	AOI_ROBOT_ACTION_GO_TO_STATION_2		:= 64,
	AOI_ROBOT_ACTION_GO_TO_ROTARY_TABLE		:= 65,
	
	AOI_ROBOT_ACTION_GO_INPUT_PRODUCT		:= 73
	
//	AOI_ROBOT_ACTION_GO_FIXTURE_TWO_PLACE	:= 65,
//	AOI_ROBOT_ACTION_GO_FIXTURE_TWO_PICK	:= 66,
//	AOI_ROBOT_ACTION_GO_FIXTURE_THREE_PLACE	:= 67,
//	AOI_ROBOT_ACTION_GO_FIXTURE_THREE_PICK	:= 68,
//	AOI_ROBOT_ACTION_GO_FIXTURE_FOUR_PLACE	:= 69,
//	AOI_ROBOT_ACTION_GO_FIXTURE_FOUR_PICK	:= 70,
//	AOI_ROBOT_ACTION_GO_TO_REJECTBOX		:= 110,
//	AOI_ROBOT_ACTION_GO_OUTPUT_PRODUCT		:= 74,
//	AOI_ROBOT_ACTION_GO_TO_GS_1				:= 120,
//	AOI_ROBOT_ACTION_GO_TO_GS_2				:= 130,
//	AOI_ROBOT_ACTION_GO_TO_GS_3				:= 140,
//	AOI_ROBOT_ACTION_GO_TO_GS_4				:= 150,
//	AOI_ROBOT_ACTION_GO_TO_GS_OUT_POSITION	:= 160,
//	AOI_ROBOT_ACTION_GO_TO_GS_LOW_2			:= 80,
//	AOI_ROBOT_ACTION_GO_TO_GS_LOW_3			:= 81,
//	AOI_ROBOT_ACTION_GO_TO_GS_LOW_4			:= 82,
//	AOI_ROBOT_ACTION_DROP					:= 300
//	AOI_ROBOT_ACTION_PICK_RNR				:= 84,
//	AOI_ROBOT_ACTION_GO_INPUT_RNR			:= 85

)UINT;
END_TYPE

// ---- POUs/Machine/Module/Robot/E_AOIRobotState.TcDUT
{attribute 'qualified_only'}
{attribute 'strict'}
TYPE E_AOIRobotState :
(
	UNINITIALIZED					:= 0,
	INITIALIZING					:= 10,
	READY_INITIALIZED				:= 20,
	IDLE							:= 30,
	PICK							:= 31,
	PLACE							:= 32,
	GO_HOME							:= 40,
	GO_BOWL							:= 45,
	GO_INPUT_PRODUCT				:= 51,
	GO_STATION_1					:= 60,
	GO_STATION_2					:= 70,
	GO_ROTARY_TABLE					:= 80,
	PLACE_ON_TABLE					:= 90,
	
	ACTION_DONE						:= 200,
	ABORT							:= -10
);
END_TYPE

// ---- POUs/Machine/Module/Robot/E_AOIRobotStateAbort.TcDUT
{attribute 'qualified_only'}
{attribute 'strict'}
TYPE E_AOIRobotStateAbort :
(
	CR800_RESET := 0,
	CR800_ABORT := 10
);
END_TYPE

// ---- POUs/Machine/Module/Robot/E_AOIRobotStateInit.TcDUT
{attribute 'qualified_only'}
{attribute 'strict'}
TYPE E_AOIRobotStateInit :
(
	CR800_RESET 	:= 0,
	CR800_INIT		:= 10
);
END_TYPE

// ---- POUs/Machine/Module/Robot/E_EtherCATStatusCheck.TcDUT
{attribute 'qualified_only'}
{attribute 'strict'}
TYPE E_EtherCATStatusCheck :
(
	MACHINE_STATE_UNINITIALIZED_CR800_ETHERCAT_STATUS_CHECK := 0,
	MACHINE_STATE_UNINITIALIZED_CR800_ETHERCAT_STATUS_CHECK_DONE := 10,
	MACHINE_STATE_UNINITIALIZED_CR800_ETHERCAT_ERROR_RESET := 20,
	MACHINE_STATE_UNINITIALIZED_CR800_ETHERCAT_REQUEST_OP_STATE := 30,
	MACHINE_STATE_UNINITIALIZED_CR800_CHECK_POWER_REGISTER := 40
);
END_TYPE

// ---- POUs/Machine/Module/RTCVision/E_RTCCameraInitState.TcDUT
{attribute 'strict'}
TYPE E_RTCCameraInitState :
(
	RTC_INIT_CONNECTION 			:= 0,
	RTC_INIT_CLEAR_BUFFER			:= 10,	
	RTC_INIT_WAIT_FOR_CONFIRMATION	:= 20,
	RTC_INIT_DONE					:= 30
);
END_TYPE

// ---- POUs/Machine/Module/RTCVision/E_RTCCameraMethodState.TcDUT
{attribute 'strict'}
TYPE E_RTCCameraMethodState :
(
	RTC_CAMERA_METHOD_SEND_COMMAND 			:= 0,
	RTC_CAMERA_METHOD_RECEIVE_RESPONSE 		:= 10
);
END_TYPE

// ---- POUs/Machine/Module/RTCVision/E_RTCCameraState.TcDUT
{attribute 'strict'}
TYPE E_RTCCameraState :
(
	RTC_CAMERA_UNINITIALIZED 				:= 0,	(* Not ready to work *)
	RTC_CAMERA_INITIALIZING					:= 10,	(* Preparing to work *)
	RTC_CAMERA_READY 						:= 20,	(* Ready to work *)
	RTC_CAMERA_IDLE							:= 30,	(* Waiting for commands *)
	RTC_CAMERA_RESET 						:= 40,	(*  *)
	
	RTC_CAMERA_SET_JOB						:= 200,	(* Set job *)
	RTC_CAMERA_START						:= 210,	(* Start job *)
	RTC_CAMERA_STOP							:= 220,	(* Stop job *)
	RTC_CAMERA_GET_RESULT					:= 230,	(* Get result *)
	RTC_CAMERA_GET_BATCH_DATA				:= 240, (* Get batch data *)
	RTC_CAMERA_CLEAR_DATA					:= 250,	(* Clear all data/parameters, prepare for new batch*)
	RTC_CAMERA_STOP_CYCLE					:= 260, (* If there is problem while production, then stop the current vision cycle, prepare a new cycle *)
	
	RTC_CAMERA_METHOD_DONE					:= 290,	(* Send command and receive confirm with vision system *)
	RTC_CAMERA_ABORTING						:= -10	(* Aborting *)
);
END_TYPE

// ---- POUs/Machine/Module/RTCVision/E_VisionJob.TcDUT
{attribute 'strict'}
{attribute 'to_string'}
TYPE E_VisionJob :
(
	UNKNOWN := 0,
	CASE_RECEIVER_E25_0100812762 := 1
);// Basic data type is INT, default initialization for all E_ColorBasic  variables is eYellow
END_TYPE

// ---- POUs/Machine/Module/RTCVision/E_VisionResult.TcDUT
{attribute 'strict'}
TYPE E_VisionResult :
(
	VISION_RESULT_UNKNOWN				:= 0,
	VISION_RESULT_GOOD 					:= 1,
	VISION_RESULT_CONTAMINATION_DIRTY	:= 2,
	VISION_RESULT_SCRATCH_DENT			:= 3,
	VISION_RESULT_REJECT				:= 4
);
END_TYPE

// ---- POUs/Machine/ST_VisuCtrlBowlFeeder.TcDUT
TYPE ST_VisuCtrlBowlFeeder :
STRUCT
	bStart : BOOL;
	bStartDisabled : BOOL;
	bStop : BOOL;
	bStopDisabled : BOOL;
	rSetpoint : REAL;
END_STRUCT
END_TYPE

// ---- VISUs/Pages/Auto/ST_SortStationParam.TcDUT
TYPE ST_SortStationParam :
STRUCT
	lrGoodPosition 		: LREAL;
	tGoodTimer			: TIME;
	
	lrDirtPosition 		: LREAL;
	tDirtTimer			: TIME;
	
	lrDentPosition 		: LREAL;
	tDentTimer			: TIME;
	
	lrRejectPosition 	: LREAL;
	tRejectTimer		: TIME;
	
END_STRUCT
END_TYPE

// ---- GVLs/GVL.TcGVL
VAR_GLOBAL CONSTANT	
	(* --- Alarm controler --- *)
	iMAX_DEFINITION_EVENTS					: UDINT := 512; 													(* Maximum size of active alarms table *)
	iMAX_EVENTS								: UDINT	:= 512; 													(* Maximum size of events table *) 
	
	(* --- Recipes manager --- *)
	iMAX_NUMBER_OF_RECIPES					: USINT 		:= 128;												(* Defines maximum number of recipes stored in recipe manager *)
	iMAX_NUMBER_OF_VARIABLES_IN_RECIPES		: USINT			:= 128;												(* Defines maximum number of parameters stored inside the recipe *)
	iMAX_RECIPE_NAME_LENGTH					: INT			:= 80;												(* Defines maximum length of the recipe name *)
	iMAX_RECIPE_DESCRIPTION_LENGTH			: INT			:= 1024;											(* Defines maximum length of the recipe description on HMI screen *)
	iMAX_RECIPE_RESTOR_BACKUP_PATH_LENGTH	: INT			:= 1024;											(* Defines maximum lenght of the path where recipes are backuped/restored *)
	sDEFAULT_RECIPE_DEFINITON				: STRING		:= 'Recipes';										(* Defines default name of recipe definition inside recipe manager *)
	sDEFAULT_LOCAL_STORAGE_PATH				: STRING(512)	:= 'C:\TwinCAT\Tests\Recipes\';						(* Defines defaul path of recipe storage *)
	
	(* --- Visu controler --- *)
	iMAX_AXIS_FRAMES						: USINT := 20;														(* Maximum frames of displayed axis in manual mode *)
	iMAX_CYLINDER_FRAMES					: USINT := 42;														(* Maximum frames of displayed cylinders in manual mode *)
	iMAX_OUTPUT_FRAMES						: USINT := 144;														(* Maximum frames of displayed outputs in manual mode *)
	iMAX_INPUT_FRAMES						: USINT := 144;														(* Maximum frames of displayed inputs in manual mode *)
	iMAX_SAFE_INPUT_FRAMES					: USINT := 36;														(* Maximum frames of displayed safe inputs in manual mode *)
	iMAX_SAFE_OUTPUT_FRAMES					: USINT := 36;														(* Maximum frames of displayed safe outputs in manual mode *)
	iMAX_ROBOT_FRAMES						: USINT := 10;														(* Maximum frames of displayed safe outputs in manual mode *)
	                                                        													
	iAXIS_PER_PAGE							: USINT := 2;														(* Number of axis displayed on single page *)
	iCYLINDERS_PER_PAGE						: USINT := 3;														(* Number of cylinders dislayed on single page *)
	iOUTPUTS_PER_PAGE						: USINT := 12;														(* Number of outputs displayed on single page *)
	iINPUTS_PER_PAGE						: USINT := 12;														(* Number of inputs displayed on single page *)
	iSAFE_INPUTS_PER_PAGE					: USINT := 6;														(* Number of safe inputs displayed on single page*)
	iSAFE_OUTPUTS_PER_PAGE					: USINT := 6;														(* Number of safe outputs displayed on single page *)
	iRECIPE_PARAMETERS_PER_PAGE				: USINT := 8;														(* Number of recipes parameters displayed on single page *)
	iROBOTS_PER_PAGE						: USINT := 1;														(* Number of recipes parameters displayed on single page *)
	
	iMAX_AXIS_PAGES							: USINT := iMAX_AXIS_FRAMES / iAXIS_PER_PAGE;						(* Defines maximum pages of axis HMI frames in manual mode *)
	iMAX_CYLINDER_PAGES						: USINT := iMAX_CYLINDER_FRAMES / iCYLINDERS_PER_PAGE;				(* Defines maximum pages of cylinders HMI frames in manual mode *)
	iMAX_OUTPUT_PAGES						: USINT := iMAX_OUTPUT_FRAMES / iOUTPUTS_PER_PAGE;					(* Defines maximum pages of digital outputs HMI frames in manual mode *)
	iMAX_INPUT_PAGES						: USINT := iMAX_INPUT_FRAMES / iINPUTS_PER_PAGE;					(* Defines maximum pages of digital inputs HMI frames in manual mode *)
	iMAX_SAFE_INPUT_PAGES					: USINT := iMAX_SAFE_INPUT_FRAMES / iSAFE_INPUTS_PER_PAGE;			(* Defines maximum pages of safe inputs HMI frames in manual mode *)
	iMAX_SAFE_OUTPUT_PAGES					: USINT := iMAX_SAFE_OUTPUT_FRAMES / iSAFE_OUTPUTS_PER_PAGE;		(* Defines maximum pages of safe outputs HMI frames in manual mode *)
	iMAX_RECIPES_PAGES						: USINT := iMAX_NUMBER_OF_RECIPES / iRECIPE_PARAMETERS_PER_PAGE;	(* Defines maximum pages of recipes parameter HMI frames in manual mode *)
	iMAX_ROBOT_PAGES						: USINT := iMAX_ROBOT_FRAMES / iROBOTS_PER_PAGE;					(* Defines maximum pages of robots HMI frames *)

	(* --- CSV Data Exchanger --- *)
	iMAX_CSV_ROWS 							: UDINT := 100;
	iMAX_CSV_COLUMNS 						: UDINT := 8;
	iMAX_CSV_FIELD_LENGTH					: UDINT := 100;
	
	(* --- Specific Machine Data --- *)
	(* Number of hardware modules *)
	iNUMBER_OF_ROBOTS							: USINT 		:= 1;//2	(* Number of robots used inside the machine *)
	
	(* --- Default machine setup --- *)
	(* Axis *)
	sROTARY_TABLE_NAME						: STRING := 'Rotary table';
	sROTARY_TABLE_MEASUREMENT_UNIT			: STRING := 'mm';
	
	(* Vision System *)
	sVISION_NAME 								: STRING 		:= 'RTC Vision System';
	sVISION_HOST 								: T_IPv4Addr 	:= '192.168.0.210';
	sVISION_AMS_NET_ID							: T_AmsNetID	:= '';
	iVISION_PORT								: UINT 			:= 23;
	tVISION_TIMEOUT								: TIME 			:= DEFAULT_ADS_TIMEOUT;
END_VAR
VAR_GLOBAL
	(* --- Library Universal Machine ---*)
	(* --- Machine data ---*)
	sMACHINE_NAME							: STRING := 'Automatic Optical Inspection Machine';					(* Full machine project name *)
	sSOFTWARE_VERSION						: STRING := '1.0.0';												(* Last taged version of control software *)
	
	(* --- Shell common features ---*)
	fbMachineTime							: FB_LocalSystemTime; 												(* Main machine clock - used by implementation of other utilites like Logger and Alarm Controler *)
	fbMachineLogger 						: FB_FileLogger; 													(* Main machine logger - registers everything that happens on machine *)

	(* --- Specific Machine ---*)
	sMACHINE_ID									: STRING		:= '35131';
	(* --- Shell Main Machine ---*)
	stShell : ST_Shell;	(* This structure contains references to Shell modules, recipe parameters and auxilary bit flags *)
	
	(* Mitsubishi robots *)
	sROBOT_NAME									: STRING		:= 'RH-3CRH4018-D-S15';
	iROBOT_OVERRIDE								: USINT			:= 100;

END_VAR

// ---- POUs/Libs/Analog Devices/Analog Device/I_AnalogDevice.TcIO
INTERFACE I_AnalogDevice

PROPERTY ModuleType : REFERENCE TO STRING
GET
END_GET
END_PROPERTY

METHOD MR_FirstCycle : BOOL
VAR_INPUT
	sName 			: STRING;
	sModuleType 	: STRING;
	sPortID			: STRING;
END_VAR
END_METHOD

PROPERTY Name : REFERENCE TO STRING
GET
END_GET
END_PROPERTY

PROPERTY PortID : REFERENCE TO STRING
GET
END_GET
END_PROPERTY

END_INTERFACE

// ---- POUs/Libs/Analog Devices/Analog Output/I_AnalogOutput.TcIO
INTERFACE I_AnalogOutput EXTENDS I_AnalogDevice

PROPERTY Value : REAL
GET
END_GET
SET
END_SET
END_PROPERTY

END_INTERFACE

// ---- POUs/Libs/Bowl Feeder/I_BowlFeeder.TcIO
INTERFACE I_BowlFeeder

PROPERTY Active : BOOL
GET
END_GET
END_PROPERTY

PROPERTY Busy : BOOL
GET
END_GET
END_PROPERTY

PROPERTY Error : BOOL
GET
END_GET
END_PROPERTY

METHOD MR_FirstCycle : BOOL
VAR_INPUT
	sName	: STRING;
END_VAR
END_METHOD

METHOD MR_Init : BOOL
VAR_INPUT
END_VAR
END_METHOD

METHOD MR_Start : BOOL
VAR_INPUT
END_VAR
END_METHOD

METHOD MR_Stop : BOOL
VAR_INPUT
END_VAR
END_METHOD

PROPERTY Running : BOOL
GET
END_GET
END_PROPERTY

PROPERTY Setpoint : REAL
GET
END_GET
SET
END_SET
END_PROPERTY

END_INTERFACE

// ---- POUs/Machine/I_MachineControl.TcIO
INTERFACE I_MachineControl EXTENDS I_UniversalMachine

PROPERTY BowlFeeder : REFERENCE TO FB_BowlFeeder
GET
END_GET
END_PROPERTY

PROPERTY Robots : REFERENCE TO FB_Robot
GET
END_GET
END_PROPERTY

PROPERTY StateInit : REFERENCE TO E_MachineCtrlStateInit
GET
END_GET
END_PROPERTY

PROPERTY StateUninitialized : REFERENCE TO E_MachineCtrlStateUninitialized
GET
END_GET
END_PROPERTY

END_INTERFACE

// ---- POUs/Machine/Module/Robot/I_AOIRobot.TcIO
INTERFACE I_AOIRobot

PROPERTY Active : BOOL
GET
END_GET
END_PROPERTY

PROPERTY Busy : BOOL
GET
END_GET
END_PROPERTY

METHOD M_EtherCATStatusCheck : BOOL
VAR_INPUT
END_VAR
END_METHOD

METHOD M_PowerOnCommand : BOOL
VAR_INPUT
END_VAR
END_METHOD

PROPERTY ModeSwitch : BOOL
SET
END_SET
END_PROPERTY

METHOD MR_Abort : BOOL
VAR_INPUT
END_VAR
END_METHOD

METHOD MR_FirstCycle : BOOL
VAR_INPUT
	sName 				: STRING;
	iInitialOverride 	: USINT;
	sPLC_NET_ID			: T_AmsNetId;
	iCR800_1_ADDRESS	: UINT;
END_VAR
END_METHOD

METHOD MR_GoBowl : BOOL
VAR_INPUT
END_VAR
END_METHOD

METHOD MR_GoHome : BOOL
VAR_INPUT
END_VAR
END_METHOD

METHOD MR_GoInputProduct : BOOL
VAR_INPUT
END_VAR
END_METHOD

METHOD MR_GoRotaryTable : BOOL
VAR_INPUT
END_VAR
END_METHOD

METHOD MR_GoStation1 : BOOL
VAR_INPUT
END_VAR
END_METHOD

METHOD MR_GoStation2 : BOOL
VAR_INPUT
END_VAR
END_METHOD

METHOD MR_Init : BOOL
VAR_INPUT
END_VAR
END_METHOD

METHOD MR_Pick : BOOL
VAR_INPUT
END_VAR
END_METHOD

METHOD MR_Place : BOOL
VAR_INPUT
END_VAR
END_METHOD

PROPERTY ref_CR800 : REFERENCE TO FB_CR800EtherCAT
GET
END_GET
END_PROPERTY

END_INTERFACE

// ---- POUs/Machine/Module/RTCVision/I_RTCVision.TcIO
INTERFACE I_RTCVision

PROPERTY Active : BOOL
GET
END_GET
END_PROPERTY

PROPERTY Busy : BOOL
GET
END_GET
END_PROPERTY

PROPERTY CurrentJob : UINT
GET
END_GET
END_PROPERTY

PROPERTY Error : BOOL
GET
END_GET
SET
END_SET
END_PROPERTY

PROPERTY ErrorID : INT
GET
END_GET
END_PROPERTY

PROPERTY JobStarted : BOOL
GET
END_GET
END_PROPERTY

PROPERTY JobStopped : BOOL
GET
END_GET
END_PROPERTY

METHOD M_CommandStation1 : BOOL
VAR_INPUT
	//PulseWidth					: TIME;
	DelayTimeForSecondTrigger	: TIME; //T#0.1ms
END_VAR
END_METHOD

METHOD M_CommandStation2 : BOOL
VAR_INPUT
	DelayTimeForSecondTrigger	: TIME; //T#0.1ms
END_VAR
END_METHOD

METHOD M_SetJob : BOOL
VAR_INPUT
	uiJob : UINT;
END_VAR
END_METHOD

METHOD M_Start : BOOL
VAR_INPUT
END_VAR
END_METHOD

METHOD M_Stop : BOOL
VAR_INPUT
END_VAR
END_METHOD

METHOD MR_FirstCycle : BOOL
VAR_INPUT	
	sName 				: STRING;
	sHost				: T_IPv4Addr;	(*  *)
	sAmsNetID 			: T_AmsNetID;	(*  *)
	iPort				: UINT;			(*  *)
	tTimeout			: TIME;			(*  *)
	
END_VAR
END_METHOD

PROPERTY Result_Station1 : UINT
GET
END_GET
END_PROPERTY

PROPERTY Result_Station2 : UINT
GET
END_GET
END_PROPERTY

END_INTERFACE

// ---- POUs/PRG/PRG_VisuControl.TcPOU
PROGRAM PRG_VisuControl
VAR
	iLoop 			: USINT;			(*  *)
	bFirstCycle 	: BOOL := TRUE;		(*  *)
	fbVisuControl	: FB_VisuControl;	(*  *)
END_VAR

IF bFirstCycle AND stShell.stFlags.bMachineCtrlAssignamentsDone 
	AND stShell.stFlags.bAlarmCtrlAssignamentsDone 
	AND stShell.stFlags.bRecipesCtrlAssignamentsDone THEN
	
	bFirstCycle := FALSE;
	
	fbVisuControl.MR_FirstCycle( 	sMachineName 		:= sMACHINE_NAME,
									sSoftwareVersion	:= sSOFTWARE_VERSION);
									
	(*--- Append platform objects to HMI ---*)
	(* Apped machine controler to HMI controler - Universal Machine Interface - Shell *)
	fbVisuControl.MR_AppendUniversalMachine(ifMachine := stShell.stPlatform.ref_fbMachineControler);
	
	(* Apped machine controler to HMI controler - FCQ Machine Interface *)
	fbVisuControl.MR_AppendAOIMachine( ifAOIMachine := stShell.stPlatform.ref_fbMachineControler);
	
	(* Append alarm controler to HMI controler *)
	fbVisuControl.MR_AppendAlarmControler(ifAlarmControler := stShell.stPlatform.ref_fbAlarmControler);
	
	(* Append recipes manager to HMI controler *)
	fbVisuControl.MR_AppendRecipesManager(ifRecipesManager := stShell.stPlatform.ref_fbRecipesManager);
	
	(* --- Append recipes parameters --- *)
	fbVisuControl.MR_AppendRecipeParameter( ifRecipeParameter := stShell.stRecipeData.rpVar1);
	fbVisuControl.MR_AppendRecipeParameter( ifRecipeParameter := stShell.stRecipeData.rpVar2);
	fbVisuControl.MR_AppendRecipeParameter( ifRecipeParameter := stShell.stRecipeData.rpVar3);
	fbVisuControl.MR_AppendRecipeParameter( ifRecipeParameter := stShell.stRecipeData.rpVar4);
	fbVisuControl.MR_AppendRecipeParameter( ifRecipeParameter := stShell.stRecipeData.rpVar5);
	fbVisuControl.MR_AppendRecipeParameter( ifRecipeParameter := stShell.stRecipeData.rpVar6);
	fbVisuControl.MR_AppendRecipeParameter( ifRecipeParameter := stShell.stRecipeData.rpVar7);
	fbVisuControl.MR_AppendRecipeParameter( ifRecipeParameter := stShell.stRecipeData.rpVar8);
	fbVisuControl.MR_AppendRecipeParameter( ifRecipeParameter := stShell.stRecipeData.rpVar9);
	fbVisuControl.MR_AppendRecipeParameter( ifRecipeParameter := stShell.stRecipeData.rpVar10);
	
	(* --- Append machine objects to HMI ---*)
//	(* Append sample digital inputs *)
//	FOR iLoop := 0 TO 19 DO
//		fbVisuControl.MR_AppendInput(ifDigitalInput := stShell.stPlatform.ref_fbMachineControler.Inputs[iLoop]);
//	END_FOR
	
//	(* Append sample digital outputs *)
//	FOR iLoop := 0 TO 19 DO
//		fbVisuControl.MR_AppendOutput(ifDigitalOutput := stShell.stPlatform.ref_fbMachineControler.Outputs[iLoop]);
//	END_FOR
	
//	(* Append sample digital inputs *)
//	FOR iLoop := 0 TO 19 DO
//		fbVisuControl.MR_AppendSafeInput(ifSafeInput := stShell.stPlatform.ref_fbMachineControler.SafeInputs[iLoop]);
//	END_FOR
	
//	(* Append sample digital outputs *)
//	FOR iLoop := 0 TO 19 DO
//		fbVisuControl.MR_AppendSafeOutput(ifSafeOutput := stShell.stPlatform.ref_fbMachineControler.SafeOutputs[iLoop]);
//	END_FOR
	
//	(* Append sample double coil cylinders *)
//	FOR iLoop := 0 TO 9 DO
//		fbVisuControl.MR_AppendCylinder( 	ifCylinder 			:= stShell.stPlatform.ref_fbMachineControler.DoubleCoilCylinders[iLoop],
//											eCylinderType 		:= CYLINDER_TYPE_DOUBLE_COIL,
//											sActiveDescription	:= 'Active',
//											sHomeDescription	:= 'Home');
//	END_FOR
	
//	(* Append sample single coil cylinders *)
//	FOR iLoop := 0 TO 9 DO
//		fbVisuControl.MR_AppendCylinder( 	ifCylinder 			:= stShell.stPlatform.ref_fbMachineControler.SingleCoilCylinders[iLoop],
//											eCylinderType 		:= CYLINDER_TYPE_SINGLE_COIL,
//											sActiveDescription 	:= 'Active',
//											sHomeDescription 	:= 'Home');
//	END_FOR
	(* Append sample scara robot *)
	//FOR iLoop := 0 TO iNUMBER_OF_ROBOTS-1 DO
		fbVisuControl.MR_AppendRobot(	ifRobot 	:= stShell.stPlatform.ref_fbMachineControler.Robots.ref_CR800,
										eRobotType	:= ROBOT_TYPE_MITSUBISHI_SCARA);
	//END_FOR
	
//	(* Append sample 6 axis robot *)
//	FOR iLoop := 5 TO 9 DO
//		fbVisuControl.MR_AppendRobot(	ifRobot 	:= stShell.stPlatform.ref_fbMachineControler.Robots[iLoop],
//										eRobotType	:= ROBOT_TYPE_MITSUBISHI_6_AXIS);
//	END_FOR
	
//	(* Append sample axes *)
//	FOR iLoop := 0 TO 19 DO
//		fbVisuControl.MR_AppendAxis(	ifMotor		:= stShell.stPlatform.ref_fbMachineControler.Axes[iLoop],
//										eMotorType	:= AXIS_TYPE_BECKHOFF_XTS_MOVER);
//	END_FOR

	(* Set assignamnet done bit *)
	stShell.stFlags.bVisuCtrlAssignamentsDone := TRUE;
END_IF

(* Start running Visu Controler if all other controlers are assigned *)
IF stShell.stFlags.bVisuCtrlAssignamentsDone THEN
	fbVisuControl();
END_IF

END_PROGRAM

// ---- POUs/Machine/FB_VisuControl.TcPOU
FUNCTION_BLOCK FB_VisuControl EXTENDS FB_UniversalVisu
VAR
	(* Page Uninitialized *)
	eUninitializedFrameSelector		: E_VisuCtrlUninitializedFrameSelector;						(* This enum is used to switch HMI frames for "Uninitialized" page *)
	stUninitializedSetupFrame 		: ST_UninitializedSetupFrame;								(* This structure contains data from "Uninitialized-Setup" page *)
	stUninitializedStartUpFrame		: ST_UninitializedStartUpFrame;								(* This structure contains data from "Uninitialized-StartUp" page *)
	
	(* Page Initializing *)                                                         	
	stInitializingFrame				: ST_InitializationFrame;									(* This structure contains data from "Initializing" page *)
	eInitializingHintFrameSelector 	: E_VisuCtrlInitializingPopUpFrameSelector;					
	bInitializingHintFrameInvisible : BOOL;		
												
	(* Common *)                  		
	ifAOIMachineCtrl		 		: I_MachineControl;	
	
	(* HMI button triggers *) 
	rtInit 							: R_TRIG;		
	rtStart							: R_TRIG;													
	rtStop							: R_TRIG;													
	ftRunning						: F_TRIG;													
	rtReset							: R_TRIG;													
	rtAbort							: R_TRIG;

	stVisuCtrlBowlFeeder : ST_VisuCtrlBowlFeeder;
END_VAR

IF bFirstCycle THEN
	(* --- Page Uninitialized --- *)
	(* Start-Up frame *)
	MEMSET(destAddr := ADR(stUninitializedStartUpFrame), fillByte := 0, n:= SIZEOF(stUninitializedStartUpFrame));
	
	(* Setup frame *)
	//Put setup frame here
	
	(* --- Page Initializing --- *)
	(* Status checkboxes reset *)
	MEMSET(destAddr := ADR(stInitializingFrame), fillByte := 0, n := SIZEOF(stInitializingFrame));
	
	(* Progress bar reset *)
	iInitProgressBar := 0;
	//iManualToAutoProgressBar := 0;
	
	(* --- Read from recipes --- *)
END_IF

(* --- Page Uninitialized --- *)
(* Wait for trigger from "Initialize" button to assign setup from HMI to Machine Controler *)
rtInit( CLK := SUPER^.btnInit);
//IF rtInit.Q THEN
	
//END_IF

(* --- Page Auto --- *)
(* Wait for trigger from "Start" button *)
rtStart( CLK := SUPER^.btnStart);

(* Wait for trigger from "Stop" button *)
rtStop( CLK := SUPER^.btnStop);

SUPER^();

METHOD M_CloseAllPopUps
VAR_INPUT
END_VAR
(* Fcq *)
F_CloseDialog('AutoPopUpStopping');
F_CloseDialog('AutoFcqPopUpTrayfeederInputEmpty');
F_CloseDialog('AutoFcqPopUpTrayfeederOutputFull');
F_CloseDialog('AutoFcqPopUpTrayfeederInterupted');
F_CloseDialog('AutoFcqPopUpCsvReaderError');
F_CloseDialog('AutoFcqPopUpInfleDeleteErrror');
F_CloseDialog('AutoFcqPopUpBatchDone');
F_CloseDialog('AutoFcqPopUpOutputTrayReplaced');
F_CloseDialog('AutoFcqPopUpRejectErrorAcknowlageInvestigate');
F_CloseDialog('AutoFcqPopUpRejectErrorCloseOutputDoors');
F_CloseDialog('AutoFcqPopUpRejectErrorContinueEject');
F_CloseDialog('AutoFcqPopUpRejectErrorRejectTrayReplaced');

(* RnR *)
F_CloseDialog('AutoRnRPopUpMissingProductInputTray');
F_CloseDialog('AutoRnRPopUpMissingProductWhileTest');
END_METHOD

METHOD MR_AppendAOIMachine : BOOL
VAR_INPUT
	ifAOIMachine : I_MachineControl;
END_VAR
THIS^.ifAOIMachineCtrl := ifAOIMachine;
MR_AppendAOIMachine := TRUE;
END_METHOD

METHOD PROTECTED MS_Aborting
SUPER^.MS_Aborting();

eUninitializedFrameSelector := VISU_CTRL_UNINITIALIZED_FRAME_STARTUP;
END_METHOD

METHOD PROTECTED MS_Auto
(* Run Shell code for "Auto" page *)
SUPER^.MS_Auto();
END_METHOD

METHOD PROTECTED  MS_Emergency
;
END_METHOD

METHOD PROTECTED MS_Initializing
(* Run Shell code for "Initializing" page *)
SUPER^.MS_Initializing();

(* --- Checkbox status update --- *)
(* Machine logger initialized *)
stInitializingFrame.bMachineLoggerInitialized := ifAOIMachineCtrl.StateInit > MACHINE_STATE_INITIALIZING_MACHINE_LOGGER;


(* Machine robots power check *)
stInitializingFrame.bRobotControlersPowerOn := ifAOIMachineCtrl.StateInit > MACHINE_STATE_INITIALIZING_ROBOTS_POWER_CHECK;

(* Robots controlers reset *)
stInitializingFrame.bRobotControlersResetDone := ifAOIMachineCtrl.StateInit > MACHINE_STATE_INITIALIZING_ROBOT_CONTROLERS_RESET;

(* Robot 1 initialized*)
stInitializingFrame.bRobotOneInitialized := ifAOIMachineCtrl.StateInit > MACHINE_STATE_INITIALIZING_ROBOT_INIT;

(* Robot 2 initialized*)
//stInitializingFrame.bRobotTwoInitialized := ifAOIMachineCtrl.StateInit > MACHINE_STATE_INITIALIZING_ROBOT_TWO_INIT;

(* Robot 1 homed *)
stInitializingFrame.bRobotOneHomed := ifAOIMachineCtrl.StateInit > MACHINE_STATE_INITIALIZING_ROBOT_HOME;

(* Robot 2 homed *)
//stInitializingFrame.bRobotTwoHomed := ifAOIMachineCtrl.StateInit > MACHINE_STATE_INITIALIZING_ROBOT_TWO_HOME;

(* Robot 1/2 in automatic mode *)
stInitializingFrame.bRobotsInAutomaticMode := ifAOIMachineCtrl.StateInit > MACHINE_STATE_INITIALIZING_ROBOT_AUTOMATIC_MODE;

(* Progress bar value update *)
iInitProgressBar := UINT_TO_USINT((STRING_TO_UINT(TO_STRING(ifAOIMachineCtrl.StateInit))*100)/STRING_TO_UINT(TO_STRING(MACHINE_STATE_INITIALIZING_DONE)));

(* User hits frame selector *)
//IF ifAOIMachineCtrl.StateInit = MACHINE_STATE_INITIALIZING_CHECK_ESTOP THEN
//	eInitializingHintFrameSelector := VISU_CTRL_INITIALIZING_FRAME_E_STOP;
//	bInitializingHintFrameInvisible := FALSE;
	
//ELSIF ifAOIMachineCtrl.StateInit = MACHINE_STATE_INITIALIZING_CHECK_DOOR_LOCKS THEN
//	eInitializingHintFrameSelector := VISU_CTRL_INITIALIZING_FRAME_DOOR_LOCK;
//	bInitializingHintFrameInvisible := FALSE;
	
//ELSIF ifAOIMachineCtrl.StateInit = MACHINE_STATE_INITIALIZING_CHECK_COURTAIN THEN
//	eInitializingHintFrameSelector := VISU_CTRL_INITIALIZING_FRAME_TRAYFEEDER_COURTAINT;
//	bInitializingHintFrameInvisible := FALSE;
	
//ELSIF ifAOIMachineCtrl.StateInit = MACHINE_STATE_INITIALIZING_SAFETY_START THEN
//	eInitializingHintFrameSelector := VISU_CTRL_INITIALIZING_FRAME_RESET_BUTTON;
//	bInitializingHintFrameInvisible := FALSE;
	
//ELSIF ifAOIMachineCtrl.StateInit = MACHINE_STATE_INITIALIZING_TRAYFEEDER_INTERUPTED_WAIT THEN
//	eInitializingHintFrameSelector := VISU_CTRL_INITIALIZING_FRAME_TRAYFEEDER_INTERUPTED;
//	bInitializingHintFrameInvisible := FALSE;
//	stInitializingFrame.stTrayfeederRetryFrame.rtTrayfeederInitRetry(CLK := stInitializingFrame.stTrayfeederRetryFrame.btnTrayfeederInitRetry);
//	IF stInitializingFrame.stTrayfeederRetryFrame.rtTrayfeederInitRetry.Q THEN
//		stInitializingFrame.stTrayfeederRetryFrame.btnTrayfeederInitRetry := FALSE;
//		ifAOIMachineCtrl.TrayfeederInitRetry := TRUE;
//	END_IF
	
//ELSIF ifAOIMachineCtrl.StateInit = MACHINE_STATE_INITIALIZING_ROTARY_TABLE_PLACE_TRAY_1 THEN
//	eInitializingHintFrameSelector := VISU_CTRL_INITIALIZING_FRAME_ROTARY_TABLE;
//	bInitializingHintFrameInvisible := FALSE;
//	stInitializingFrame.stRotaryTableFrame.rtContinue(CLK := stInitializingFrame.stRotaryTableFrame.btnContinue);
//	IF stInitializingFrame.stRotaryTableFrame.rtContinue.Q THEN
//		stInitializingFrame.stRotaryTableFrame.btnContinue := FALSE;
//		ifAOIMachineCtrl.InitRotate := TRUE;
//	END_IF
	
//ELSIF ifAOIMachineCtrl.StateInit = MACHINE_STATE_INITIALIZING_ROTARY_TABLE_PLACE_TRAY_2 THEN
//	eInitializingHintFrameSelector := VISU_CTRL_INITIALIZING_FRAME_ROTARY_TABLE;
//	bInitializingHintFrameInvisible := FALSE;
//	stInitializingFrame.stRotaryTableFrame.rtContinue(CLK := stInitializingFrame.stRotaryTableFrame.btnContinue);
//	IF stInitializingFrame.stRotaryTableFrame.rtContinue.Q THEN
//		stInitializingFrame.stRotaryTableFrame.btnContinue := FALSE;
//		ifAOIMachineCtrl.InitRotate := TRUE;
//	END_IF
	
//ELSIF ifAOIMachineCtrl.StateInit = MACHINE_STATE_INITIALIZING_FIRST_FIXTURE_INIT_FAILED OR
//		ifAOIMachineCtrl.StateInit = MACHINE_STATE_INITIALIZING_SECOND_FIXTURE_INIT_FAILED OR
//		ifAOIMachineCtrl.StateInit = MACHINE_STATE_INITIALIZING_THIRD_FIXTURE_INIT_FAILED OR
//		ifAOIMachineCtrl.StateInit = MACHINE_STATE_INITIALIZING_FOURTH_FIXTURE_INIT_FAILED OR
//		ifAOIMachineCtrl.StateInit = MACHINE_STATE_INITIALIZING_FIFTH_FIXTURE_INIT_FAILED OR
//		ifAOIMachineCtrl.StateInit = MACHINE_STATE_INITIALIZING_SIXTH_FIXTURE_INIT_FAILED OR
//		ifAOIMachineCtrl.StateInit = MACHINE_STATE_INITIALIZING_SEVENTH_FIXTURE_INIT_FAILED OR
//		ifAOIMachineCtrl.StateInit = MACHINE_STATE_INITIALIZING_EIGHT_FIXTURE_INIT_FAILED THEN
//		eInitializingHintFrameSelector := VISU_CTRL_INITIALIZING_FRAME_FIXTURE_CONNECTION_FAILED;
//		bInitializingHintFrameInvisible := FALSE;
		
//		stInitializingFrame.stFixtureFailedFrame.rtFixtureInitRetry(CLK := stInitializingFrame.stFixtureFailedFrame.btnFixtureInitRetry);
//		stInitializingFrame.stFixtureFailedFrame.rtFixtureInitSkip(CLK := stInitializingFrame.stFixtureFailedFrame.btnFixtureInitSkip);
//		IF stInitializingFrame.stFixtureFailedFrame.rtFixtureInitRetry.Q THEN
//			stInitializingFrame.stFixtureFailedFrame.btnFixtureInitRetry := FALSE;
//			ifAOIMachineCtrl.FixtureInitRetry := TRUE;
//		ELSIF stInitializingFrame.stFixtureFailedFrame.rtFixtureInitSkip.Q THEN
//			stInitializingFrame.stFixtureFailedFrame.btnFixtureInitSkip := FALSE;
//			ifAOIMachineCtrl.FixtureInitSkip := TRUE;
//		END_IF
	
//ELSIF ifAOIMachineCtrl.StateInit = MACHINE_STATE_INITIALIZING_FIXTURES_INIT_FAILED THEN
//	eInitializingHintFrameSelector := VISU_CTRL_INITIALIZING_FRAME_NO_FIXTURES_AVAILABLE;
//	bInitializingHintFrameInvisible := FALSE;
	
//ELSE
//	bInitializingHintFrameInvisible := TRUE;
//END_IF
END_METHOD

METHOD PROTECTED MS_Uninitialized
(* Run Shell code for "Uninitialized" page *)
SUPER^.MS_Uninitialized();

M_CloseAllPopUps();

CASE eUninitializedFrameSelector OF
	VISU_CTRL_UNINITIALIZED_FRAME_STARTUP:
		eCurrentNavigation := NAVIGATION_EMPTY;
		
		(* Power on robot controlers *)
		stUninitializedStartUpFrame.bCR800PowerOn := ifAOIMachineCtrl.StateUninitialized > MACHINE_STATE_UNINITIALIZED_CR800_CHECK_POWER_REGISTER;
		stUninitializedStartUpFrame.bCR800EtherCatInitialization := ifAOIMachineCtrl.StateUninitialized > MACHINE_STATE_UNINITIALIZED_CR800_CHECK_POWER_REGISTER;

		(* Progress bar value update *)
		stUninitializedStartUpFrame.iProgressBar := (STRING_TO_USINT(TO_STRING(ifAOIMachineCtrl.StateUninitialized))*100)/60;
		
		(* Start-Up finished -> switch frame *)
		IF ifAOIMachineCtrl.StateUninitialized = MACHINE_STATE_UNINITIALIZED_DONE THEN
			eUninitializedFrameSelector := VISU_CTRL_UNINITIALIZED_FRAME_SETUP;
			eCurrentNavigation := NAVIGATION_UNINITIALIZED;
		END_IF
	
	VISU_CTRL_UNINITIALIZED_FRAME_SETUP:
		;
		
END_CASE
END_METHOD

END_FUNCTION_BLOCK

// ---- POUs/Libs/Platform/Universal Visu/FB_UniversalVisu.TcPOU
(* 
:Description: This function block is base for of machine HMI module in all projects.
*)
FUNCTION_BLOCK ABSTRACT FB_UniversalVisu
VAR
	(* --- Auxilary variables --- *)
	bFirstCycle 						: BOOL := TRUE;	(*  *)
	iLoop								: USINT;		(*  *)
	iLoop2								: USINT;		(*  *)
	                        			
	(* --- Header --- *)    			
	sMachineName						: STRING;	(*  *)
	sSoftwareVersion					: STRING;	(*  *)
	sCurrentDate						: STRING;	(*  *)
	sCurrentTime						: STRING;	(*  *)
	sCurrentUser						: STRING;	(*  *)
	sCurrentRecipe						: STRING;	(*  *)
                            			
	iActiveAlarms						: UDINT;				(*  *)
	iActiveCriticals 					: REFERENCE TO UDINT;	(*  *)
	iActvieErrors						: REFERENCE TO UDINT;	(*  *)
	iActiveWarrnings					: REFERENCE TO UDINT;	(*  *)
	
	(* --- Navigation bar --- *)
	btnInit								: BOOL;		(*  *)
	btnReset							: BOOL;		(*  *)
	btnManual 							: BOOL;		(*  *)
	btnAuto								: BOOL;		(*  *)
	btnAbort 							: BOOL;		(*  *)
	btnStart 							: BOOL;		(*  *)
	btnStop 							: BOOL;		(*  *)
	btnStepMode 						: BOOL;		(*  *)
	btnBack 							: BOOL;		(*  *)
	                    			
	bInit								: BOOL;		(*  *)
	bReset								: BOOL;		(*  *)
	bAbort 								: BOOL;		(*  *)
	
	(* --- Auxilary navigation bar --- *)
	btnCloseHMI							: BOOL;		(*  *)
	btnAlarms							: BOOL;		(*  *)
	btnRecipes							: BOOL;		(*  *)
	btnLogIn							: BOOL;		(*  *)
	btnLogOut							: BOOL;		(*  *)
	btnChangePass						: BOOL;		(*  *)
	btnLights							: BOOL;		(*  *)
	                        			
	sCloseHMIFileName					: STRING := 'C:\Windows\System32\cmd.exe';	(*  *) //'C:\HMI Utility\CloseHMI.bat',
	sCloseHMIParameters					: STRING := 'taskkill /IM Tc3PlcHmi.exe /F';	(*  *) //'C:\HMI Utility',
	
	(* --- Initialization indicators --- *)
	iInitProgressBar 					: USINT;			(*  *)
	
	(* --- Manual mode --- *)	
	btnManualCylinder					: BOOL;				(*  *)
	btnManualAxis						: BOOL;				(*  *)
	btnManualSafety						: BOOL;				(*  *)
	btnManualOthers						: BOOL;				(*  *)
	btnManualOutputs					: BOOL;				(*  *)
	btnManualInputs						: BOOL;				(*  *)
	btnManualRobots						: BOOL;				(*  *)
	                        			
	bManualCylinderDisabled				: BOOL := FALSE;	(*  *)
	bManualAxisDisabled					: BOOL := FALSE;	(*  *)
	bManualInputsDisabled				: BOOL := FALSE;	(*  *)
	bManualOutputsDisabled				: BOOL := FALSE;	(*  *)
	bManualSafetyDisabled				: BOOL := FALSE;	(*  *)
	bManualOthersDisabled				: BOOL := FALSE;	(*  *)
	bManualRobotDisabled				: BOOL := FALSE;	(*  *)	
	
	btnNext								: BOOL;			(* *)
	btnPrevious							: BOOL;			(* *)
	btnNextInput						: BOOL;			(* *)
	btnPreviousInput					: BOOL;			(* *)
	btnNextOutput						: BOOL;			(* *)
	btnPreviousOutput					: BOOL;			(*  *)
                                    	
	bNextInvisible						: BOOL;			(*  *)
	bPreviousInvisible					: BOOL;			(*  *)
	bNextInvisibleInput					: BOOL;			(*  *)
	bPreviousInvisibleInput				: BOOL;			(*  *)
	bNextInvisibleOutput				: BOOL;			(*  *)
	bPreviousInvisibleOutput			: BOOL;			(*  *)
	                                	
	iSelectedCylinderPageIndex			: USINT := 0;	(*  *)
	iSelectedAxisPageIndex				: USINT := 0;	(*  *)
	iSelectedInputPageIndex 			: USINT := 0;	(*  *)
	iSelectedOutputPageIndex			: USINT := 0;	(*  *)
	iSelectedSafeInputPageIndex 		: USINT := 0;	(*  *)
	iSelectedSafeOutputPageIndex		: USINT := 0;	(*  *)
	iSelectedRobotPageIndex				: USINT := 0;	(*  *)
	
	iCylinderIndex						: USINT := 0;	(*  *)
	iAxisIndex							: USINT := 0;	(*  *)
	iInputIndex							: USINT := 0;	(*  *)
	iOutputIndex						: USINT := 0;	(*  *)
	iSafeInputIndex						: USINT := 0;	(*  *)
	iSafeOutputIndex					: USINT := 0;	(*  *)
	iRobotIndex							: USINT := 0;	(*  *)
                            			
	iCylinderPageIndex					: USINT := 0;	(*  *)
	iAxisPageIndex						: USINT := 0;	(*  *)
	iInputPageIndex						: USINT := 0;	(*  *)
	iOutputPageIndex					: USINT := 0;	(*  *)
	iSafeInputPageIndex					: USINT := 0;	(*  *)
	iSafeOutputPageIndex				: USINT := 0;	(*  *)
	iRobotPageIndex						: USINT := 0;	(*  *)
	                        			
	iCylinderFrameIndex					: USINT := 0;	(*  *)
	iAxisFrameIndex						: USINT := 0;	(*  *)
	iInputFrameIndex					: USINT := 0;	(*  *)
	iOutputFrameIndex					: USINT := 0;	(*  *)
	iSafeInputFrameIndex				: USINT := 0;	(*  *)
	iSafeOutputFrameIndex				: USINT := 0;	(*  *)
	iRobotFrameIndex					: USINT := 0;	(*  *)
                            			
	arrCylinderFrameEmpty 				: ARRAY [0..iMAX_CYLINDER_PAGES-1] OF ARRAY [0..iCYLINDERS_PER_PAGE-1] OF BOOL;								(*  *)
	arrAxisFrameEmpty					: ARRAY [0..iMAX_AXIS_PAGES-1] OF ARRAY [0..iAXIS_PER_PAGE-1] OF BOOL;										(*  *)
	arrInputFrameEmpty					: ARRAY [0..iMAX_INPUT_PAGES-1] OF ARRAY [0..iINPUTS_PER_PAGE-1] OF BOOL;									(*  *)
	arrOutputFrameEmpty					: ARRAY [0..iMAX_OUTPUT_PAGES-1] OF ARRAY [0..iOUTPUTS_PER_PAGE-1] OF BOOL;									(*  *)
	arrSafeInputFrameEmpty				: ARRAY [0..iMAX_SAFE_INPUT_PAGES-1] OF ARRAY [0..iSAFE_INPUTS_PER_PAGE-1] OF BOOL;							(*  *)
	arrSafeOutputFrameEmpty				: ARRAY [0..iMAX_SAFE_OUTPUT_PAGES-1] OF ARRAY [0..iSAFE_OUTPUTS_PER_PAGE-1] OF BOOL;						(*  *)
	arrRobotFrameEmpty					: ARRAY [0..iMAX_ROBOT_PAGES-1] OF ARRAY [0..iROBOTS_PER_PAGE-1] OF BOOL;									(*  *)
	                        			
	arrCylinderFrame					: ARRAY [0..iMAX_CYLINDER_PAGES-1] OF ARRAY [0..iCYLINDERS_PER_PAGE-1] OF ST_VisuCtrlCylinderFrame;			(*  *)
	arrAxisFrame						: ARRAY [0..iMAX_AXIS_PAGES-1] OF ARRAY [0..iAXIS_PER_PAGE-1] OF ST_VisuCtrlAxisFrame;						(*  *)
	arrInputFrame						: ARRAY [0..iMAX_INPUT_PAGES-1] OF ARRAY [0..iINPUTS_PER_PAGE-1] OF ST_VisuCtrlInputFrame;					(*  *)
	arrOutputFrame						: ARRAY [0..iMAX_OUTPUT_PAGES-1] OF ARRAY [0..iOUTPUTS_PER_PAGE-1] OF ST_VisuCtrlOutputFrame;				(*  *)
	arrSafeInputFrame					: ARRAY	[0..iMAX_SAFE_INPUT_PAGES-1] OF ARRAY [0..iSAFE_INPUTS_PER_PAGE-1] OF ST_VisuCtrlInputFrame;		(*  *)
	arrSafeOutputFrame					: ARRAY [0..iMAX_SAFE_OUTPUT_PAGES-1] OF ARRAY [0..iSAFE_OUTPUTS_PER_PAGE-1] OF ST_VisuCtrlOutputFrame;		(*  *)
	arrRobotFrame						: ARRAY [0..iMAX_ROBOT_PAGES-1] OF ARRAY [0..iROBOTS_PER_PAGE-1] OF ST_VisuCtrlRobotFrame;					(*  *)
		                    			
	arrCylinderState					: ARRAY [0..iMAX_CYLINDER_PAGES-1] OF ARRAY [0..iCYLINDERS_PER_PAGE-1] OF E_VisuCtrlSingleCylinderState;	(*  *)
	arrAxisState						: ARRAY [0..iMAX_AXIS_PAGES-1] OF ARRAY [0..iAXIS_PER_PAGE-1] OF E_VisuCtrlSingleAxisState;					(*  *)
	arrRobotState						: ARRAY [0..iMAX_ROBOT_PAGES-1] OF ARRAY [0..iROBOTS_PER_PAGE-1] OF E_VisuCtrlSingleRobotState;				(*  *)
                            			
